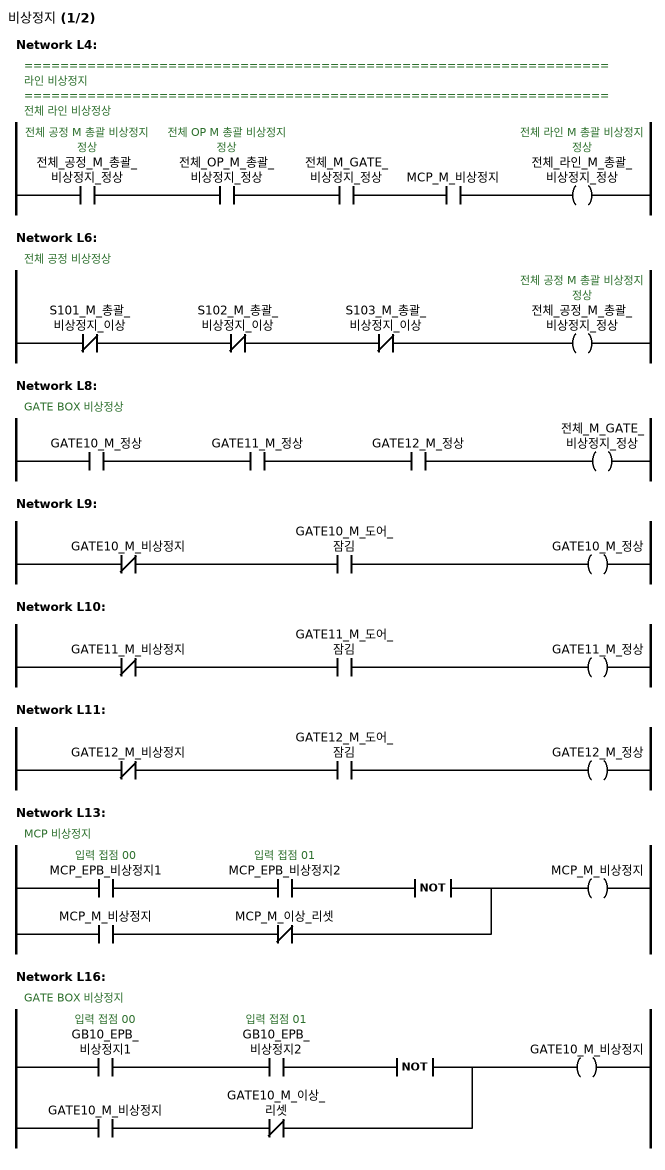
(* ================================================================= *)
(* 라인 비상정지 *)
(* ================================================================= *)
(* 전체 라인 비상정상 *)
(* Rung L4 *)
전체_라인_M_총괄_비상정지_정상 := 전체_공정_M_총괄_비상정지_정상 AND 전체_OP_M_총괄_비상정지_정상 AND 전체_M_GATE_비상정지_정상 AND MCP_M_비상정지;
(* 전체 공정 비상정상 *)
(* Rung L6 *)
전체_공정_M_총괄_비상정지_정상 := NOT S101_M_총괄_비상정지_이상 AND NOT S102_M_총괄_비상정지_이상 AND NOT S103_M_총괄_비상정지_이상;
(* GATE BOX 비상정상 *)
(* Rung L8 *)
전체_M_GATE_비상정지_정상 := GATE10_M_정상 AND GATE11_M_정상 AND GATE12_M_정상;
(* Rung L9 *)
GATE10_M_정상 := NOT GATE10_M_비상정지 AND GATE10_M_도어_잠김;
(* Rung L10 *)
GATE11_M_정상 := NOT GATE11_M_비상정지 AND GATE11_M_도어_잠김;
(* Rung L11 *)
GATE12_M_정상 := NOT GATE12_M_비상정지 AND GATE12_M_도어_잠김;
(* MCP 비상정지 *)
(* Rung L13 *)
MCP_M_비상정지 := NOT (MCP_EPB_비상정지1 AND MCP_EPB_비상정지2) OR (MCP_M_비상정지 AND NOT MCP_M_이상_리셋);
(* GATE BOX 비상정지 *)
(* Rung L16 *)
GATE10_M_비상정지 := NOT (GB10_EPB_비상정지1 AND GB10_EPB_비상정지2) OR (GATE10_M_비상정지 AND NOT GATE10_M_이상_리셋);

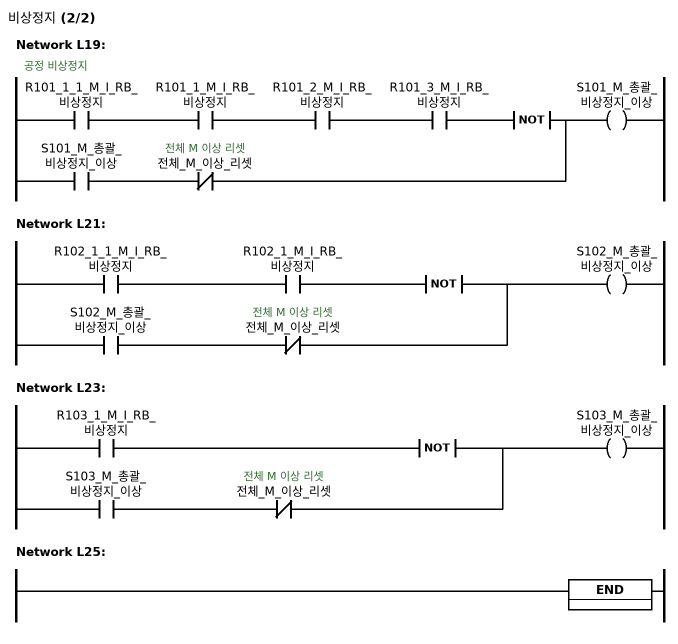
(* 공정 비상정지 *)
(* Rung L19 *)
S101_M_총괄_비상정지_이상 := NOT (R101_1_1_M_I_RB_비상정지 AND R101_1_M_I_RB_비상정지 AND R101_2_M_I_RB_비상정지 AND R101_3_M_I_RB_비상정지) OR (S101_M_총괄_비상정지_이상 AND NOT 전체_M_이상_리셋);
(* Rung L21 *)
S102_M_총괄_비상정지_이상 := NOT (R102_1_1_M_I_RB_비상정지 AND R102_1_M_I_RB_비상정지) OR (S102_M_총괄_비상정지_이상 AND NOT 전체_M_이상_리셋);
(* Rung L23 *)
S103_M_총괄_비상정지_이상 := NOT R103_1_M_I_RB_비상정지 OR (S103_M_총괄_비상정지_이상 AND NOT 전체_M_이상_리셋);
(* Rung L25 *)
END();
END_PROGRAM

PROGRAM S101_유틸리티 (* task: 스캔 프로그램 *)
VAR_EXTERNAL
    AWAYS_ON : BOOL; (* AT %MW3.1 *)
    EGIS_EJS : BOOL;
    MCP_PBL_101_자동_운전 : BOOL; (* AT %MW87630.4 *) (* 입력 접점 04 *)
    MCP_PBL_운전준비_ON : BOOL; (* AT %MW87630.0 *) (* 입력 접점 00 *)
    MCP_SSP_101_수동_선택 : BOOL; (* AT %MW87630.2 *) (* 입력 접점 02 *)
    MCP_SSP_101_자동_선택 : BOOL; (* AT %MW87630.3 *) (* 입력 접점 03 *)
    R101_1_1_M_I_RB_2차_작업완료 : BOOL; (* AT %MW20041.3 *)
    R101_1_1_M_I_RB_간섭무_1 : BOOL; (* AT %MW20042.0 *)
    R101_1_1_M_I_RB_간섭무_2 : BOOL; (* AT %MW20042.1 *)
    R101_1_1_M_I_RB_원위치 : BOOL; (* AT %MW20040.3 *)
    R101_1_1_M_SEQ : WORD; (* AT %MW10000 *) (* R101_1_1_M_SEQ *)
    R101_1_1_M_STN_차종_NONE : BOOL; (* AT %MW1002.3 *)
    R101_1_1_M_STN_차종_ON : BOOL; (* AT %MW1002.2 *)
    R101_1_1_M_차종1_AX : BOOL; (* AT %MW10001.0 *) (* R101_1_1_M_차종1_AX *)
    R101_1_1_M_차종1_B : BOOL; (* AT %MW10001.1 *) (* R101_1_1_M_차종1_B *)
    R101_1_1_M_차종1_C : BOOL; (* AT %MW10001.2 *) (* R101_1_1_M_차종1_C *)
    R101_1_1_M_차종1_D : BOOL; (* AT %MW10001.3 *) (* R101_1_1_M_차종1_D *)
    R101_1_1_M_차종1_E : BOOL; (* AT %MW10001.4 *) (* R101_1_1_M_차종1_E *)
    R101_1_1_M_차종1_F : BOOL; (* AT %MW10001.5 *) (* R101_1_1_M_차종1_F *)
    R101_1_1_M_차종1_G : BOOL; (* AT %MW10001.6 *) (* R101_1_1_M_차종1_G *)
    R101_1_1_M_차종1_H : BOOL; (* AT %MW10001.7 *) (* R101_1_1_M_차종1_H *)
    R101_1_1_M_차종2_3DR : BOOL; (* AT %MW10001.8 *) (* R101_1_1_M_차종2_3DR *)
    R101_1_1_M_차종2_4DR : BOOL; (* AT %MW10001.9 *) (* R101_1_1_M_차종2_4DR *)
    R101_1_1_M_차종2_5DR : BOOL; (* AT %MW10001.10 *) (* R101_1_1_M_차종2_5DR *)
    R101_1_1_M_차종2_SP1 : BOOL; (* AT %MW10001.12 *) (* R101_1_1_M_차종2_SP1 *)
    R101_1_1_M_차종2_SP2 : BOOL; (* AT %MW10001.13 *) (* R101_1_1_M_차종2_SP2 *)
    R101_1_1_M_차종2_WGN : BOOL; (* AT %MW10001.11 *) (* R101_1_1_M_차종2_WGN *)
    R101_1_1_M_차종3_LHD : BOOL; (* AT %MW10001.14 *) (* R101_1_1_M_차종3_LHD *)
    R101_1_1_M_차종3_RHD : BOOL; (* AT %MW10001.15 *) (* R101_1_1_M_차종3_RHD *)
    R101_1_1_M_차종4_EEC : BOOL; (* AT %MW10002.3 *) (* R101_1_1_M_차종4_EEC *)
    R101_1_1_M_차종4_SP1 : BOOL; (* AT %MW10002.8 *) (* R101_1_1_M_차종4_SP1 *)
    R101_1_1_M_차종4_SP2 : BOOL; (* AT %MW10002.9 *) (* R101_1_1_M_차종4_SP2 *)
    R101_1_1_M_차종4_SP3 : BOOL; (* AT %MW10002.11 *) (* R101_1_1_M_차종4_SP3 *)
    R101_1_1_M_차종4_SP4 : BOOL; (* AT %MW10002.12 *) (* R101_1_1_M_차종4_SP4 *)
    R101_1_1_M_차종4_SP5 : BOOL; (* AT %MW10002.13 *) (* R101_1_1_M_차종4_SP5 *)
    R101_1_1_M_차종4_SP6 : BOOL; (* AT %MW10002.14 *) (* R101_1_1_M_차종4_SP6 *)
    R101_1_1_M_차종4_SP7 : BOOL; (* AT %MW10002.15 *) (* R101_1_1_M_차종4_SP7 *)
    R101_1_1_M_차종4_내수 : BOOL; (* AT %MW10002.0 *) (* R101_1_1_M_차종4_내수 *)
    R101_1_1_M_차종4_러시아 : BOOL; (* AT %MW10002.10 *) (* R101_1_1_M_차종4_러시아 *)
    R101_1_1_M_차종4_북미 : BOOL; (* AT %MW10002.2 *) (* R101_1_1_M_차종4_북미 *)
    R101_1_1_M_차종4_브라질 : BOOL; (* AT %MW10002.7 *) (* R101_1_1_M_차종4_브라질 *)
    R101_1_1_M_차종4_수출 : BOOL; (* AT %MW10002.1 *) (* R101_1_1_M_차종4_수출 *)
    R101_1_1_M_차종4_중국 : BOOL; (* AT %MW10002.6 *) (* R101_1_1_M_차종4_중국 *)
    R101_1_1_M_차종4_중동 : BOOL; (* AT %MW10002.5 *) (* R101_1_1_M_차종4_중동 *)
    R101_1_1_M_차종4_호주 : BOOL; (* AT %MW10002.4 *) (* R101_1_1_M_차종4_호주 *)
    R101_1_1_M_차종5_AT : BOOL; (* AT %MW10003.1 *) (* R101_1_1_M_차종5_AT *)
    R101_1_1_M_차종5_MT : BOOL; (* AT %MW10003.0 *) (* R101_1_1_M_차종5_MT *)
    R101_1_1_M_차종5_SP1 : BOOL; (* AT %MW10003.2 *) (* R101_1_1_M_차종5_SP1 *)
    R101_1_1_M_차종6_DSROOF : BOOL; (* AT %MW10003.6 *) (* R101_1_1_M_차종6_DSROOF *)
    R101_1_1_M_차종6_SP1 : BOOL; (* AT %MW10003.7 *) (* R101_1_1_M_차종6_SP1 *)
    R101_1_1_M_차종6_썬루프 : BOOL; (* AT %MW10003.4 *) (* R101_1_1_M_차종6_썬루프 *)
    R101_1_1_M_차종6_일반루프 : BOOL; (* AT %MW10003.3 *) (* R101_1_1_M_차종6_일반루프 *)
    R101_1_1_M_차종6_파노라마루프 : BOOL; (* AT %MW10003.5 *) (* R101_1_1_M_차종6_파노라마루프 *)
    R101_1_1_M_차종7_DSL : BOOL; (* AT %MW10003.9 *) (* R101_1_1_M_차종7_DSL *)
    R101_1_1_M_차종7_GSL : BOOL; (* AT %MW10003.8 *) (* R101_1_1_M_차종7_GSL *)
    R101_1_1_M_차종7_SP1 : BOOL; (* AT %MW10003.10 *) (* R101_1_1_M_차종7_SP1 *)
    R101_1_1_M_차종7_SP2 : BOOL; (* AT %MW10003.11 *) (* R101_1_1_M_차종7_SP2 *)
    R101_1_1_M_차종7_SP3 : BOOL; (* AT %MW10003.12 *) (* R101_1_1_M_차종7_SP3 *)
    R101_1_1_M_차종7_SP4 : BOOL; (* AT %MW10003.13 *) (* R101_1_1_M_차종7_SP4 *)
    R101_1_1_M_차종7_SP5 : BOOL; (* AT %MW10003.14 *) (* R101_1_1_M_차종7_SP5 *)
    R101_1_1_M_차종7_SP6 : BOOL; (* AT %MW10003.15 *) (* R101_1_1_M_차종7_SP6 *)
    R101_1_1_M_차종8_2WD : BOOL; (* AT %MW10004.0 *) (* R101_1_1_M_차종8_2WD *)
    R101_1_1_M_차종8_4WD : BOOL; (* AT %MW10004.1 *) (* R101_1_1_M_차종8_4WD *)
    R101_1_1_M_차종8_SP1 : BOOL; (* AT %MW10004.2 *) (* R101_1_1_M_차종8_SP1 *)
    R101_1_1_M_차종9_MPI : BOOL; (* AT %MW10004.3 *) (* R101_1_1_M_차종9_MPI *)
    R101_1_1_M_차종9_SP1 : BOOL; (* AT %MW10004.5 *) (* R101_1_1_M_차종9_SP1 *)
    R101_1_1_M_차종9_SP10 : BOOL; (* AT %MW10004.14 *) (* R101_1_1_M_차종9_SP10 *)
    R101_1_1_M_차종9_SP11 : BOOL; (* AT %MW10004.15 *) (* R101_1_1_M_차종9_SP11 *)
    R101_1_1_M_차종9_SP2 : BOOL; (* AT %MW10004.6 *) (* R101_1_1_M_차종9_SP2 *)
    R101_1_1_M_차종9_SP3 : BOOL; (* AT %MW10004.7 *) (* R101_1_1_M_차종9_SP3 *)
    R101_1_1_M_차종9_SP4 : BOOL; (* AT %MW10004.8 *) (* R101_1_1_M_차종9_SP4 *)
    R101_1_1_M_차종9_SP5 : BOOL; (* AT %MW10004.9 *) (* R101_1_1_M_차종9_SP5 *)
    R101_1_1_M_차종9_SP6 : BOOL; (* AT %MW10004.10 *) (* R101_1_1_M_차종9_SP6 *)
    R101_1_1_M_차종9_SP7 : BOOL; (* AT %MW10004.11 *) (* R101_1_1_M_차종9_SP7 *)
    R101_1_1_M_차종9_SP8 : BOOL; (* AT %MW10004.12 *) (* R101_1_1_M_차종9_SP8 *)
    R101_1_1_M_차종9_SP9 : BOOL; (* AT %MW10004.13 *) (* R101_1_1_M_차종9_SP9 *)
    R101_1_1_M_차종9_T_GDI : BOOL; (* AT %MW10004.4 *) (* R101_1_1_M_차종9_T_GDI *)
    R101_1_1_M_차종_OPT1_R_RACK_무 : BOOL; (* AT %MW10005.3 *) (* R101_1_1_M_차종_OPT1_R_RACK_무 *)
    R101_1_1_M_차종_OPT1_R_RACK_유 : BOOL; (* AT %MW10005.2 *) (* R101_1_1_M_차종_OPT1_R_RACK_유 *)
    R101_1_1_M_차종_OPT1_SP1 : BOOL; (* AT %MW10005.10 *) (* R101_1_1_M_차종_OPT1_SP1 *)
    R101_1_1_M_차종_OPT1_SP2 : BOOL; (* AT %MW10005.11 *) (* R101_1_1_M_차종_OPT1_SP2 *)
    R101_1_1_M_차종_OPT1_SP3 : BOOL; (* AT %MW10005.12 *) (* R101_1_1_M_차종_OPT1_SP3 *)
    R101_1_1_M_차종_OPT1_SP4 : BOOL; (* AT %MW10005.13 *) (* R101_1_1_M_차종_OPT1_SP4 *)
    R101_1_1_M_차종_OPT1_SP5 : BOOL; (* AT %MW10005.14 *) (* R101_1_1_M_차종_OPT1_SP5 *)
    R101_1_1_M_차종_OPT1_SP6 : BOOL; (* AT %MW10005.15 *) (* R101_1_1_M_차종_OPT1_SP6 *)
    R101_1_1_M_차종_OPT1_S_REP_EATER_무 : BOOL; (* AT %MW10005.7 *) (* R101_1_1_M_차종_OPT1_S_REP_EATER_무 *)
    R101_1_1_M_차종_OPT1_S_REP_EATER_유 : BOOL; (* AT %MW10005.6 *) (* R101_1_1_M_차종_OPT1_S_REP_EATER_유 *)
    R101_1_1_M_차종_OPT1_VAN_무 : BOOL; (* AT %MW10005.9 *) (* R101_1_1_M_차종_OPT1_VAN_무 *)
    R101_1_1_M_차종_OPT1_VAN_유 : BOOL; (* AT %MW10005.8 *) (* R101_1_1_M_차종_OPT1_VAN_유 *)
    R101_1_1_M_차종_OPT1_슬라이딩_무 : BOOL; (* AT %MW10005.1 *) (* R101_1_1_M_차종_OPT1_슬라이딩_무 *)
    R101_1_1_M_차종_OPT1_슬라이딩_유 : BOOL; (* AT %MW10005.0 *) (* R101_1_1_M_차종_OPT1_슬라이딩_유 *)
    R101_1_1_M_차종_OPT1_폴딩_무 : BOOL; (* AT %MW10005.5 *) (* R101_1_1_M_차종_OPT1_폴딩_무 *)
    R101_1_1_M_차종_OPT1_폴딩_유 : BOOL; (* AT %MW10005.4 *) (* R101_1_1_M_차종_OPT1_폴딩_유 *)
    R101_1_M_I_RB_간섭무_2 : BOOL; (* AT %MW20072.1 *)
    R101_1_M_I_RB_원위치 : BOOL; (* AT %MW20070.3 *)
    R101_1_M_I_RB_최종작업완료 : BOOL; (* AT %MW20071.0 *)
    R101_1_M_RB_PROG_NO : WORD; (* AT %MW20074 *)
    R101_2_M_I_RB_간섭무_2 : BOOL; (* AT %MW20062.1 *)
    R101_2_M_I_RB_원위치 : BOOL; (* AT %MW20060.3 *)
    R101_2_M_I_RB_최종작업완료 : BOOL; (* AT %MW20061.0 *)
    R101_3_M_I_RB_간섭무_2 : BOOL; (* AT %MW20052.1 *)
    R101_3_M_I_RB_원위치 : BOOL; (* AT %MW20050.3 *)
    R102_1_M_I_RB_2차_작업완료 : BOOL; (* AT %MW20081.3 *)
    R102_1_M_I_RB_3차_작업완료 : BOOL; (* AT %MW20081.4 *)
    R102_1_M_I_RB_4차_작업완료 : BOOL; (* AT %MW20081.5 *)
    R102_1_M_I_RB_간섭무_1 : BOOL; (* AT %MW20082.0 *)
    R102_1_M_I_RB_간섭무_2 : BOOL; (* AT %MW20082.1 *)
    R102_1_M_I_RB_간섭무_3 : BOOL; (* AT %MW20082.2 *)
    R102_1_M_I_RB_원위치 : BOOL; (* AT %MW20080.3 *)
    R103_1_M_I_RB_최종작업완료 : BOOL; (* AT %MW20101.0 *)
    S101_3축_1_운전준비1 : BOOL; (* AT %MW50000.0 *)
    S101_3축_1_운전준비2 : BOOL; (* AT %MW50000.1 *)
    S101_3축_1_이상_리셋 : BOOL; (* AT %MW51000.7 *)
    S101_3축_2_운전준비1 : BOOL; (* AT %MW50100.0 *)
    S101_3축_2_운전준비2 : BOOL; (* AT %MW50100.1 *)
    S101_3축_2_이상_리셋 : BOOL; (* AT %MW51100.7 *)
    S101_3축_3_FAULT : BOOL; (* AT %MW50200.3 *)
    S101_3축_3_운전준비1 : BOOL; (* AT %MW50200.0 *)
    S101_3축_3_운전준비2 : BOOL; (* AT %MW50200.1 *)
    S101_3축_3_이상_리셋 : BOOL; (* AT %MW51200.7 *)
    S101_MCR_비상정지1 : BOOL; (* AT %MW95207.0 *) (* 출력 접점 00 *)
    S101_MCR_비상정지2 : BOOL; (* AT %MW95207.1 *) (* 출력 접점 01 *)
    S101_MCR_비상정지3 : BOOL; (* AT %MW95207.2 *) (* 출력 접점 02 *)
    S101_M_3_축1_전진단 : BOOL; (* AT %MW1102.3 *)
    S101_M_3_축1_후진단 : BOOL; (* AT %MW1102.4 *)
    S101_M_3_축2_전진단 : BOOL; (* AT %MW1103.3 *)
    S101_M_3_축2_후진단 : BOOL; (* AT %MW1103.4 *)
    S101_M_3_축3_전진단 : BOOL; (* AT %MW1104.3 *)
    S101_M_3_축3_후진단 : BOOL; (* AT %MW1104.4 *)
    S101_M_APRON_LH_안착OK_POS : BOOL; (* AT %MW1004.8 *)
    S101_M_APRON_RH_안착OK_POS : BOOL; (* AT %MW1004.9 *)
    S101_M_AX_래치_전진단 : BOOL; (* AT %MW1100.3 *)
    S101_M_AX_래치_후진단 : BOOL; (* AT %MW1100.4 *)
    S101_M_DASH_안착OK_POS : BOOL; (* AT %MW1004.10 *)
    S101_M_DASH_클램프_전진단 : BOOL; (* AT %MW1105.3 *)
    S101_M_DASH_클램프_후진단 : BOOL; (* AT %MW1105.4 *)
    S101_M_FRT_취출OK_POS : BOOL; (* AT %MW1004.11 *)
    S101_M_SEQ : WORD; (* AT %MW10020 *) (* S101_M_SEQ *)
    S101_M_SHIFT_전진단 : BOOL; (* AT %MW1101.3 *)
    S101_M_SHIFT_후진단 : BOOL; (* AT %MW1101.4 *)
    S101_M_STN_DASH_로딩완료 : BOOL; (* AT %MW1001.12 *)
    S101_M_STN_FRT_FLR_취출완료 : BOOL; (* AT %MW1001.13 *)
    S101_M_STN_LH_로딩완료 : BOOL; (* AT %MW1001.10 *)
    S101_M_STN_RH_로딩완료 : BOOL; (* AT %MW1001.11 *)
    S101_M_STN_차종_NONE : BOOL; (* AT %MW1002.1 *)
    S101_M_STN_차종_ON : BOOL; (* AT %MW1002.0 *)
    S101_M_공정_APRON_제품감지_OFF : BOOL; (* AT %MW1001.4 *)
    S101_M_공정_APRON_제품감지_ON : BOOL; (* AT %MW1001.3 *)
    S101_M_공정_DASH_제품감지_OFF : BOOL; (* AT %MW1001.6 *)
    S101_M_공정_DASH_제품감지_ON : BOOL; (* AT %MW1001.5 *)
    S101_M_공정_HOME_POSI : BOOL; (* AT %MW1004.0 *)
    S101_M_공정_간섭무 : BOOL; (* AT %MW1004.1 *)
    S101_M_공정_사양감지_OK : BOOL; (* AT %MW1001.7 *)
    S101_M_사양이상 : BOOL; (* AT %MW1019.0 *)
    S101_M_수동_모드 : BOOL; (* AT %MW1000.3 *)
    S101_M_운전준비_ON : BOOL; (* AT %MW1000.0 *)
    S101_M_자동_START : BOOL; (* AT %MW1000.5 *)
    S101_M_자동_모드 : BOOL; (* AT %MW1000.1 *)
    S101_M_자동_운전중 : BOOL; (* AT %MW1000.4 *)
    S101_M_작업_완료 : BOOL; (* AT %MW1001.0 *)
    S101_M_작업_완료_보조 : BOOL; (* AT %MW1000.9 *)
    S101_M_전체_클램프_잠김단 : BOOL; (* AT %MW1004.12 *)
    S101_M_차종1_AX : BOOL; (* AT %MW10021.0 *) (* S101_M_차종1_AX *)
    S101_M_차종1_B : BOOL; (* AT %MW10021.1 *) (* S101_M_차종1_B *)
    S101_M_차종1_C : BOOL; (* AT %MW10021.2 *) (* S101_M_차종1_C *)
    S101_M_차종1_D : BOOL; (* AT %MW10021.3 *) (* S101_M_차종1_D *)
    S101_M_차종1_E : BOOL; (* AT %MW10021.4 *) (* S101_M_차종1_E *)
    S101_M_차종1_F : BOOL; (* AT %MW10021.5 *) (* S101_M_차종1_F *)
    S101_M_차종1_G : BOOL; (* AT %MW10021.6 *) (* S101_M_차종1_G *)
    S101_M_차종1_H : BOOL; (* AT %MW10021.7 *) (* S101_M_차종1_H *)
    S101_M_차종2_3DR : BOOL; (* AT %MW10021.8 *) (* S101_M_차종2_3DR *)
    S101_M_차종2_4DR : BOOL; (* AT %MW10021.9 *) (* S101_M_차종2_4DR *)
    S101_M_차종2_5DR : BOOL; (* AT %MW10021.10 *) (* S101_M_차종2_5DR *)
    S101_M_차종2_SP1 : BOOL; (* AT %MW10021.12 *) (* S101_M_차종2_SP1 *)
    S101_M_차종2_SP2 : BOOL; (* AT %MW10021.13 *) (* S101_M_차종2_SP2 *)
    S101_M_차종2_WGN : BOOL; (* AT %MW10021.11 *) (* S101_M_차종2_WGN *)
    S101_M_차종3_LHD : BOOL; (* AT %MW10021.14 *) (* S101_M_차종3_LHD *)
    S101_M_차종3_RHD : BOOL; (* AT %MW10021.15 *) (* S101_M_차종3_RHD *)
    S101_M_차종4_EEC : BOOL; (* AT %MW10022.3 *) (* S101_M_차종4_EEC *)
    S101_M_차종4_SP1 : BOOL; (* AT %MW10022.8 *) (* S101_M_차종4_SP1 *)
    S101_M_차종4_SP2 : BOOL; (* AT %MW10022.9 *) (* S101_M_차종4_SP2 *)
    S101_M_차종4_SP3 : BOOL; (* AT %MW10022.11 *) (* S101_M_차종4_SP3 *)
    S101_M_차종4_SP4 : BOOL; (* AT %MW10022.12 *) (* S101_M_차종4_SP4 *)
    S101_M_차종4_SP5 : BOOL; (* AT %MW10022.13 *) (* S101_M_차종4_SP5 *)
    S101_M_차종4_SP6 : BOOL; (* AT %MW10022.14 *) (* S101_M_차종4_SP6 *)
    S101_M_차종4_SP7 : BOOL; (* AT %MW10022.15 *) (* S101_M_차종4_SP7 *)
    S101_M_차종4_내수 : BOOL; (* AT %MW10022.0 *) (* S101_M_차종4_내수 *)
    S101_M_차종4_러시아 : BOOL; (* AT %MW10022.10 *) (* S101_M_차종4_러시아 *)
    S101_M_차종4_북미 : BOOL; (* AT %MW10022.2 *) (* S101_M_차종4_북미 *)
    S101_M_차종4_브라질 : BOOL; (* AT %MW10022.7 *) (* S101_M_차종4_브라질 *)
    S101_M_차종4_수출 : BOOL; (* AT %MW10022.1 *) (* S101_M_차종4_수출 *)
    S101_M_차종4_중국 : BOOL; (* AT %MW10022.6 *) (* S101_M_차종4_중국 *)
    S101_M_차종4_중동 : BOOL; (* AT %MW10022.5 *) (* S101_M_차종4_중동 *)
    S101_M_차종4_호주 : BOOL; (* AT %MW10022.4 *) (* S101_M_차종4_호주 *)
    S101_M_차종5_AT : BOOL; (* AT %MW10023.1 *) (* S101_M_차종5_AT *)
    S101_M_차종5_MT : BOOL; (* AT %MW10023.0 *) (* S101_M_차종5_MT *)
    S101_M_차종5_SP1 : BOOL; (* AT %MW10023.2 *) (* S101_M_차종5_SP1 *)
    S101_M_차종6_DSROOF : BOOL; (* AT %MW10023.6 *) (* S101_M_차종6_DSROOF *)
    S101_M_차종6_SP1 : BOOL; (* AT %MW10023.7 *) (* S101_M_차종6_SP1 *)
    S101_M_차종6_썬루프 : BOOL; (* AT %MW10023.4 *) (* S101_M_차종6_썬루프 *)
    S101_M_차종6_일반루프 : BOOL; (* AT %MW10023.3 *) (* S101_M_차종6_일반루프 *)
    S101_M_차종6_파노라마루프 : BOOL; (* AT %MW10023.5 *) (* S101_M_차종6_파노라마루프 *)
    S101_M_차종7_DSL : BOOL; (* AT %MW10023.9 *) (* S101_M_차종7_DSL *)
    S101_M_차종7_GSL : BOOL; (* AT %MW10023.8 *) (* S101_M_차종7_GSL *)
    S101_M_차종7_SP1 : BOOL; (* AT %MW10023.10 *) (* S101_M_차종7_SP1 *)
    S101_M_차종7_SP2 : BOOL; (* AT %MW10023.11 *) (* S101_M_차종7_SP2 *)
    S101_M_차종7_SP3 : BOOL; (* AT %MW10023.12 *) (* S101_M_차종7_SP3 *)
    S101_M_차종7_SP4 : BOOL; (* AT %MW10023.13 *) (* S101_M_차종7_SP4 *)
    S101_M_차종7_SP5 : BOOL; (* AT %MW10023.14 *) (* S101_M_차종7_SP5 *)
    S101_M_차종7_SP6 : BOOL; (* AT %MW10023.15 *) (* S101_M_차종7_SP6 *)
    S101_M_차종8_2WD : BOOL; (* AT %MW10024.0 *) (* S101_M_차종8_2WD *)
    S101_M_차종8_4WD : BOOL; (* AT %MW10024.1 *) (* S101_M_차종8_4WD *)
    S101_M_차종8_SP1 : BOOL; (* AT %MW10024.2 *) (* S101_M_차종8_SP1 *)
    S101_M_차종9_MPI : BOOL; (* AT %MW10024.3 *) (* S101_M_차종9_MPI *)
    S101_M_차종9_SP1 : BOOL; (* AT %MW10024.5 *) (* S101_M_차종9_SP1 *)
    S101_M_차종9_SP10 : BOOL; (* AT %MW10024.14 *) (* S101_M_차종9_SP10 *)
    S101_M_차종9_SP11 : BOOL; (* AT %MW10024.15 *) (* S101_M_차종9_SP11 *)
    S101_M_차종9_SP2 : BOOL; (* AT %MW10024.6 *) (* S101_M_차종9_SP2 *)
    S101_M_차종9_SP3 : BOOL; (* AT %MW10024.7 *) (* S101_M_차종9_SP3 *)
    S101_M_차종9_SP4 : BOOL; (* AT %MW10024.8 *) (* S101_M_차종9_SP4 *)
    S101_M_차종9_SP5 : BOOL; (* AT %MW10024.9 *) (* S101_M_차종9_SP5 *)
    S101_M_차종9_SP6 : BOOL; (* AT %MW10024.10 *) (* S101_M_차종9_SP6 *)
    S101_M_차종9_SP7 : BOOL; (* AT %MW10024.11 *) (* S101_M_차종9_SP7 *)
    S101_M_차종9_SP8 : BOOL; (* AT %MW10024.12 *) (* S101_M_차종9_SP8 *)
    S101_M_차종9_SP9 : BOOL; (* AT %MW10024.13 *) (* S101_M_차종9_SP9 *)
    S101_M_차종9_T_GDI : BOOL; (* AT %MW10024.4 *) (* S101_M_차종9_T_GDI *)
    S101_M_차종_OPT1_R_RACK_무 : BOOL; (* AT %MW10025.3 *) (* S101_M_차종_OPT1_R_RACK_무 *)
    S101_M_차종_OPT1_R_RACK_유 : BOOL; (* AT %MW10025.2 *) (* S101_M_차종_OPT1_R_RACK_유 *)
    S101_M_차종_OPT1_SP1 : BOOL; (* AT %MW10025.10 *) (* S101_M_차종_OPT1_SP1 *)
    S101_M_차종_OPT1_SP2 : BOOL; (* AT %MW10025.11 *) (* S101_M_차종_OPT1_SP2 *)
    S101_M_차종_OPT1_SP3 : BOOL; (* AT %MW10025.12 *) (* S101_M_차종_OPT1_SP3 *)
    S101_M_차종_OPT1_SP4 : BOOL; (* AT %MW10025.13 *) (* S101_M_차종_OPT1_SP4 *)
    S101_M_차종_OPT1_SP5 : BOOL; (* AT %MW10025.14 *) (* S101_M_차종_OPT1_SP5 *)
    S101_M_차종_OPT1_SP6 : BOOL; (* AT %MW10025.15 *) (* S101_M_차종_OPT1_SP6 *)
    S101_M_차종_OPT1_S_REP_EATER_무 : BOOL; (* AT %MW10025.7 *) (* S101_M_차종_OPT1_S_REP_EATER_무 *)
    S101_M_차종_OPT1_S_REP_EATER_유 : BOOL; (* AT %MW10025.6 *) (* S101_M_차종_OPT1_S_REP_EATER_유 *)
    S101_M_차종_OPT1_VAN_무 : BOOL; (* AT %MW10025.9 *) (* S101_M_차종_OPT1_VAN_무 *)
    S101_M_차종_OPT1_VAN_유 : BOOL; (* AT %MW10025.8 *) (* S101_M_차종_OPT1_VAN_유 *)
    S101_M_차종_OPT1_슬라이딩_무 : BOOL; (* AT %MW10025.1 *) (* S101_M_차종_OPT1_슬라이딩_무 *)
    S101_M_차종_OPT1_슬라이딩_유 : BOOL; (* AT %MW10025.0 *) (* S101_M_차종_OPT1_슬라이딩_유 *)
    S101_M_차종_OPT1_폴딩_무 : BOOL; (* AT %MW10025.5 *) (* S101_M_차종_OPT1_폴딩_무 *)
    S101_M_차종_OPT1_폴딩_유 : BOOL; (* AT %MW10025.4 *) (* S101_M_차종_OPT1_폴딩_유 *)
    S101_M_핀클램프_전진단 : BOOL; (* AT %MW1106.3 *)
    S101_M_핀클램프_후진단 : BOOL; (* AT %MW1106.4 *)
    S101_PRS_I_3축_DASH_파트1_ON : BOOL; (* AT %MW86102.6 *) (* 입력 접점 06 *)
    S101_PRS_I_3축_DASH_파트2_ON : BOOL; (* AT %MW86102.7 *) (* 입력 접점 07 *)
    S101_PRS_I_3축_LH_파트_ON : BOOL; (* AT %MW86102.4 *) (* 입력 접점 04 *)
    S101_PRS_I_3축_RH_파트_ON : BOOL; (* AT %MW86102.5 *) (* 입력 접점 05 *)
    S101_PRS_I_AX_APRON_LHD_사양감지 : BOOL; (* AT %MW86102.8 *)
    S101_PRS_I_AX_APRON_RHD_사양감지 : BOOL; (* AT %MW86102.9 *)
    S101_PRS_I_AX_DASH_파트_ON : BOOL; (* AT %MW86102.2 *)
    S101_PRS_I_AX_LH_파트_ON : BOOL; (* AT %MW86102.0 *)
    S101_PRS_I_AX_RH_파트_ON : BOOL; (* AT %MW86102.1 *)
    S101_운전준비 : TON;
    S103_M_공정_제품감지_ON : BOOL; (* AT %MW2001.3 *)
    T101_자동 : TON;
    전체_M_GATE_자동기동 : BOOL; (* AT %MW308.1 *) (* 전체 M GATE 자동기동 *)
    전체_M_이상_리셋 : BOOL; (* AT %MW308.2 *) (* 전체 M 이상 리셋 *)
    전체_라인_M_총괄_SAFETY_이상 : BOOL; (* AT %MW300.2 *)
    전체_라인_M_총괄_공기압_이상 : BOOL; (* AT %MW300.3 *)
    전체_라인_M_총괄_비상정지_이상 : BOOL; (* AT %MW300.1 *)
    전체_라인_M_총괄_이상 : BOOL; (* AT %MW300.0 *)
END_VAR
VAR
    _R101_1_RB_비교_PROG_NO : INT;
    작업_COMP : TON;
END_VAR
VAR
    _t1 : BOOL;
    _t2 : BOOL;
    _t3 : BOOL;
    _t4 : BOOL;
    _p5 : BOOL;
END_VAR

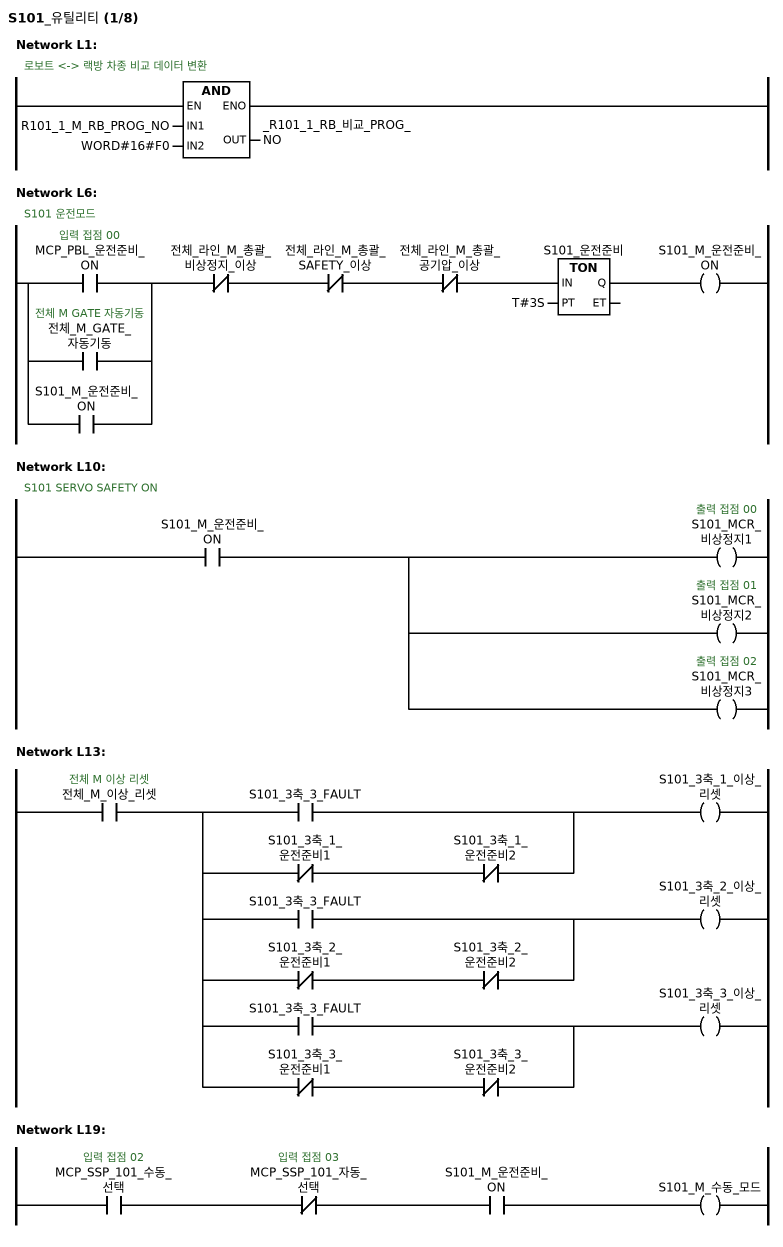
(* 로보트 <-> 랙방 차종 비교 데이터 변환 *)
(* Rung L1 *)
_R101_1_RB_비교_PROG_NO := R101_1_M_RB_PROG_NO AND WORD#16#F0;
(* S101 운전모드 *)
(* Rung L6 *)
S101_운전준비(IN := (MCP_PBL_운전준비_ON OR 전체_M_GATE_자동기동 OR S101_M_운전준비_ON) AND NOT 전체_라인_M_총괄_비상정지_이상 AND NOT 전체_라인_M_총괄_SAFETY_이상 AND NOT 전체_라인_M_총괄_공기압_이상, PT := T#3S);
S101_M_운전준비_ON := S101_운전준비.Q;
(* S101 SERVO SAFETY ON *)
(* Rung L10 *)
S101_MCR_비상정지1 := S101_M_운전준비_ON;
S101_MCR_비상정지2 := S101_M_운전준비_ON;
S101_MCR_비상정지3 := S101_M_운전준비_ON;
(* Rung L13 *)
S101_3축_1_이상_리셋 := 전체_M_이상_리셋 AND (S101_3축_3_FAULT OR (NOT S101_3축_1_운전준비1 AND NOT S101_3축_1_운전준비2));
S101_3축_2_이상_리셋 := 전체_M_이상_리셋 AND (S101_3축_3_FAULT OR (NOT S101_3축_2_운전준비1 AND NOT S101_3축_2_운전준비2));
S101_3축_3_이상_리셋 := 전체_M_이상_리셋 AND (S101_3축_3_FAULT OR (NOT S101_3축_3_운전준비1 AND NOT S101_3축_3_운전준비2));
(* Rung L19 *)
S101_M_수동_모드 := MCP_SSP_101_수동_선택 AND NOT MCP_SSP_101_자동_선택 AND S101_M_운전준비_ON;

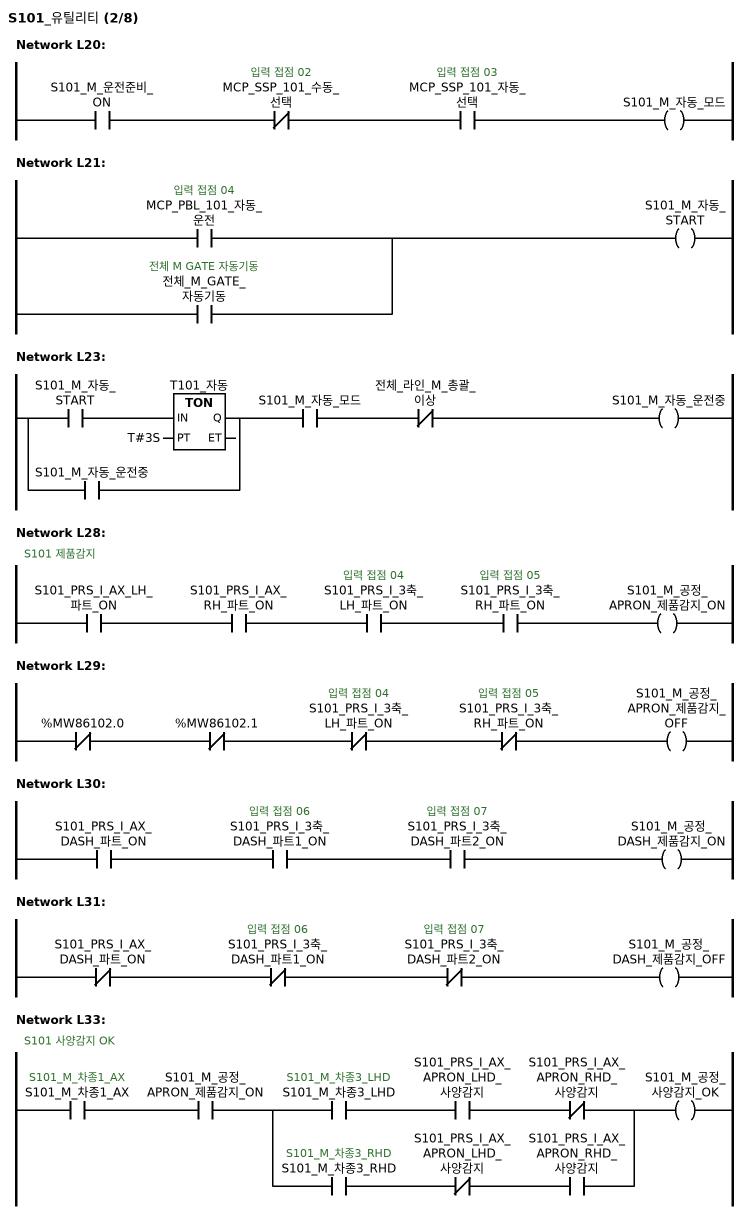
(* Rung L20 *)
S101_M_자동_모드 := S101_M_운전준비_ON AND NOT MCP_SSP_101_수동_선택 AND MCP_SSP_101_자동_선택;
(* Rung L21 *)
S101_M_자동_START := MCP_PBL_101_자동_운전 OR 전체_M_GATE_자동기동;
(* Rung L23 *)
T101_자동(IN := S101_M_자동_START, PT := T#3S);
S101_M_자동_운전중 := (T101_자동.Q OR S101_M_자동_운전중) AND S101_M_자동_모드 AND NOT 전체_라인_M_총괄_이상;
(* S101 제품감지 *)
(* Rung L28 *)
S101_M_공정_APRON_제품감지_ON := S101_PRS_I_AX_LH_파트_ON AND S101_PRS_I_AX_RH_파트_ON AND S101_PRS_I_3축_LH_파트_ON AND S101_PRS_I_3축_RH_파트_ON;
(* Rung L29 *)
S101_M_공정_APRON_제품감지_OFF := NOT %MW86102.0 AND NOT %MW86102.1 AND NOT S101_PRS_I_3축_LH_파트_ON AND NOT S101_PRS_I_3축_RH_파트_ON;
(* Rung L30 *)
S101_M_공정_DASH_제품감지_ON := S101_PRS_I_AX_DASH_파트_ON AND S101_PRS_I_3축_DASH_파트1_ON AND S101_PRS_I_3축_DASH_파트2_ON;
(* Rung L31 *)
S101_M_공정_DASH_제품감지_OFF := NOT S101_PRS_I_AX_DASH_파트_ON AND NOT S101_PRS_I_3축_DASH_파트1_ON AND NOT S101_PRS_I_3축_DASH_파트2_ON;
(* S101 사양감지 OK *)
(* Rung L33 *)
S101_M_공정_사양감지_OK := S101_M_차종1_AX AND S101_M_공정_APRON_제품감지_ON AND ((S101_M_차종3_LHD AND S101_PRS_I_AX_APRON_LHD_사양감지 AND NOT S101_PRS_I_AX_APRON_RHD_사양감지) OR (S101_M_차종3_RHD AND NOT S101_PRS_I_AX_APRON_LHD_사양감지 AND S101_PRS_I_AX_APRON_RHD_사양감지));

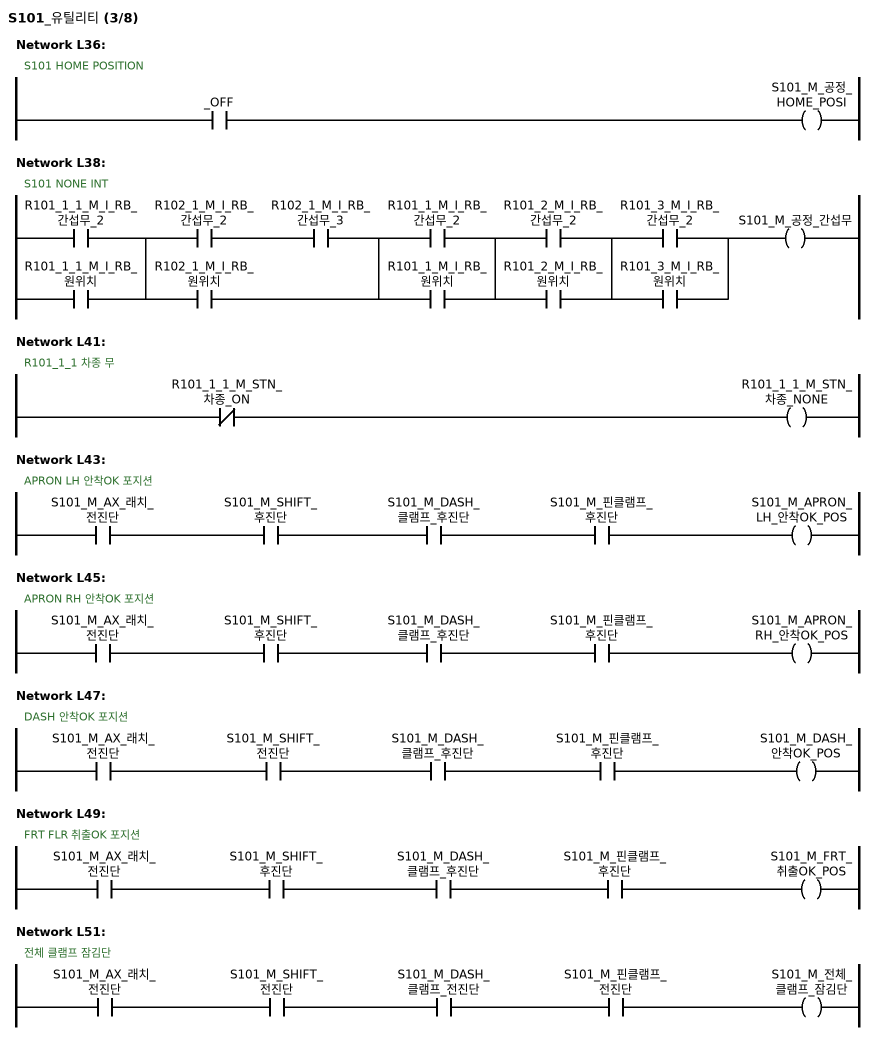
(* S101 HOME POSITION *)
(* Rung L36 *)
S101_M_공정_HOME_POSI := _OFF;
(* S101 NONE INT *)
(* Rung L38 *)
S101_M_공정_간섭무 := (R101_1_1_M_I_RB_간섭무_2 OR R101_1_1_M_I_RB_원위치) AND ((R102_1_M_I_RB_간섭무_2 AND R102_1_M_I_RB_간섭무_3) OR R102_1_M_I_RB_원위치) AND (R101_1_M_I_RB_간섭무_2 OR R101_1_M_I_RB_원위치) AND (R101_2_M_I_RB_간섭무_2 OR R101_2_M_I_RB_원위치) AND (R101_3_M_I_RB_간섭무_2 OR R101_3_M_I_RB_원위치);
(* R101_1_1 차종 무 *)
(* Rung L41 *)
R101_1_1_M_STN_차종_NONE := NOT R101_1_1_M_STN_차종_ON;
(* APRON LH 안착OK 포지션 *)
(* Rung L43 *)
S101_M_APRON_LH_안착OK_POS := S101_M_AX_래치_전진단 AND S101_M_SHIFT_후진단 AND S101_M_DASH_클램프_후진단 AND S101_M_핀클램프_후진단;
(* APRON RH 안착OK 포지션 *)
(* Rung L45 *)
S101_M_APRON_RH_안착OK_POS := S101_M_AX_래치_전진단 AND S101_M_SHIFT_후진단 AND S101_M_DASH_클램프_후진단 AND S101_M_핀클램프_후진단;
(* DASH 안착OK 포지션 *)
(* Rung L47 *)
S101_M_DASH_안착OK_POS := S101_M_AX_래치_전진단 AND S101_M_SHIFT_전진단 AND S101_M_DASH_클램프_후진단 AND S101_M_핀클램프_후진단;
(* FRT FLR 취출OK 포지션 *)
(* Rung L49 *)
S101_M_FRT_취출OK_POS := S101_M_AX_래치_전진단 AND S101_M_SHIFT_후진단 AND S101_M_DASH_클램프_후진단 AND S101_M_핀클램프_후진단;
(* 전체 클램프 잠김단 *)
(* Rung L51 *)
S101_M_전체_클램프_잠김단 := S101_M_AX_래치_전진단 AND S101_M_SHIFT_전진단 AND S101_M_DASH_클램프_전진단 AND S101_M_핀클램프_전진단;

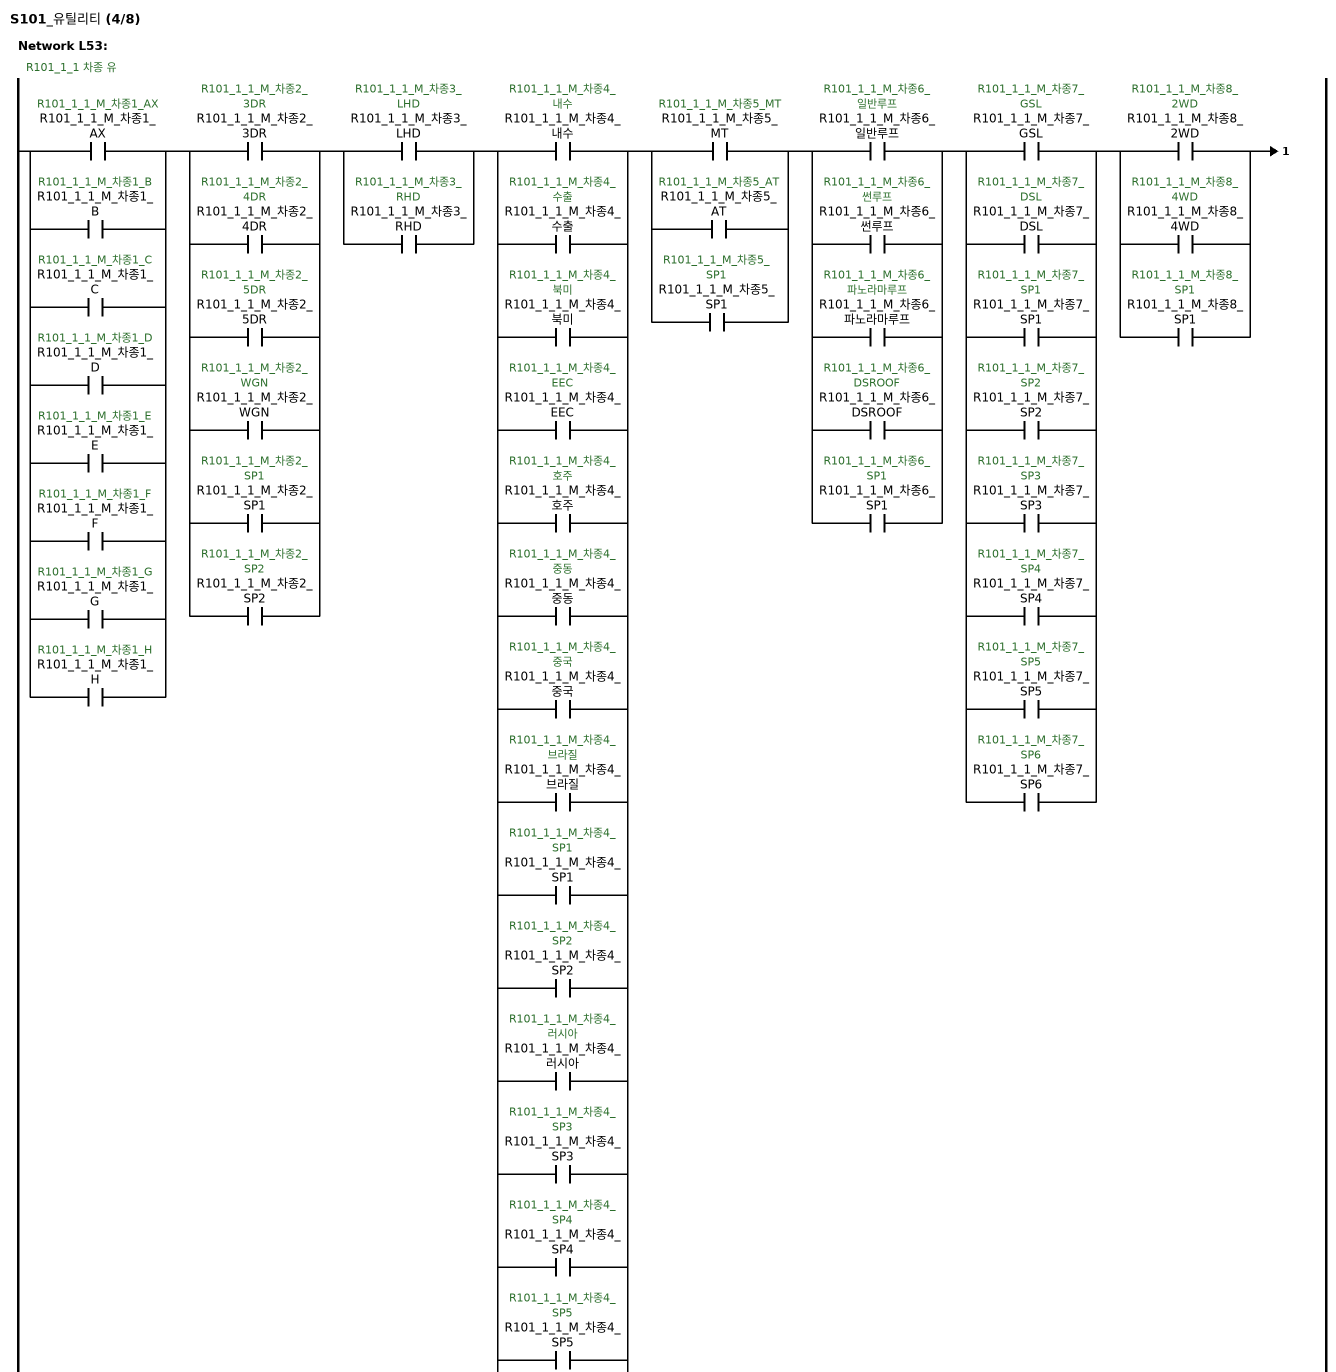

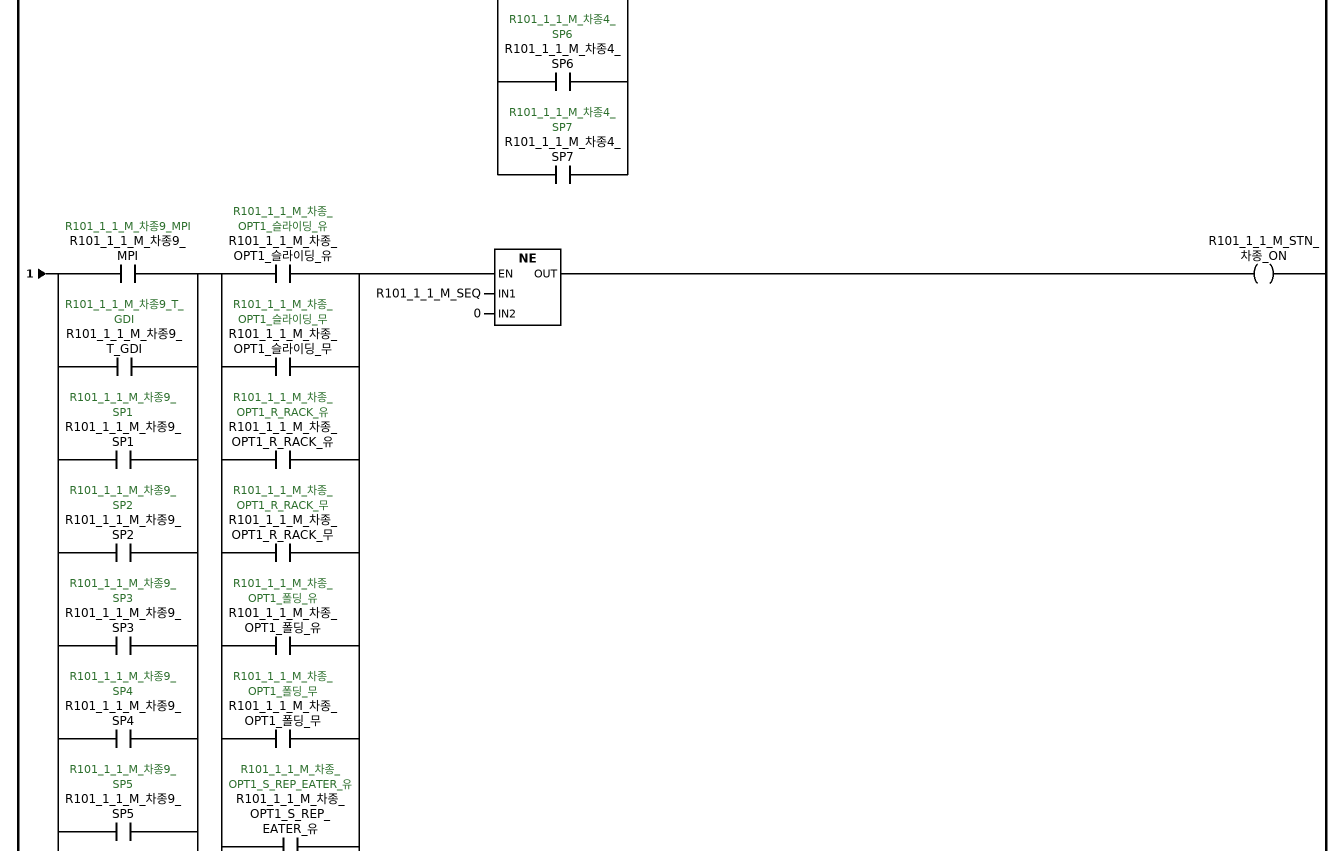

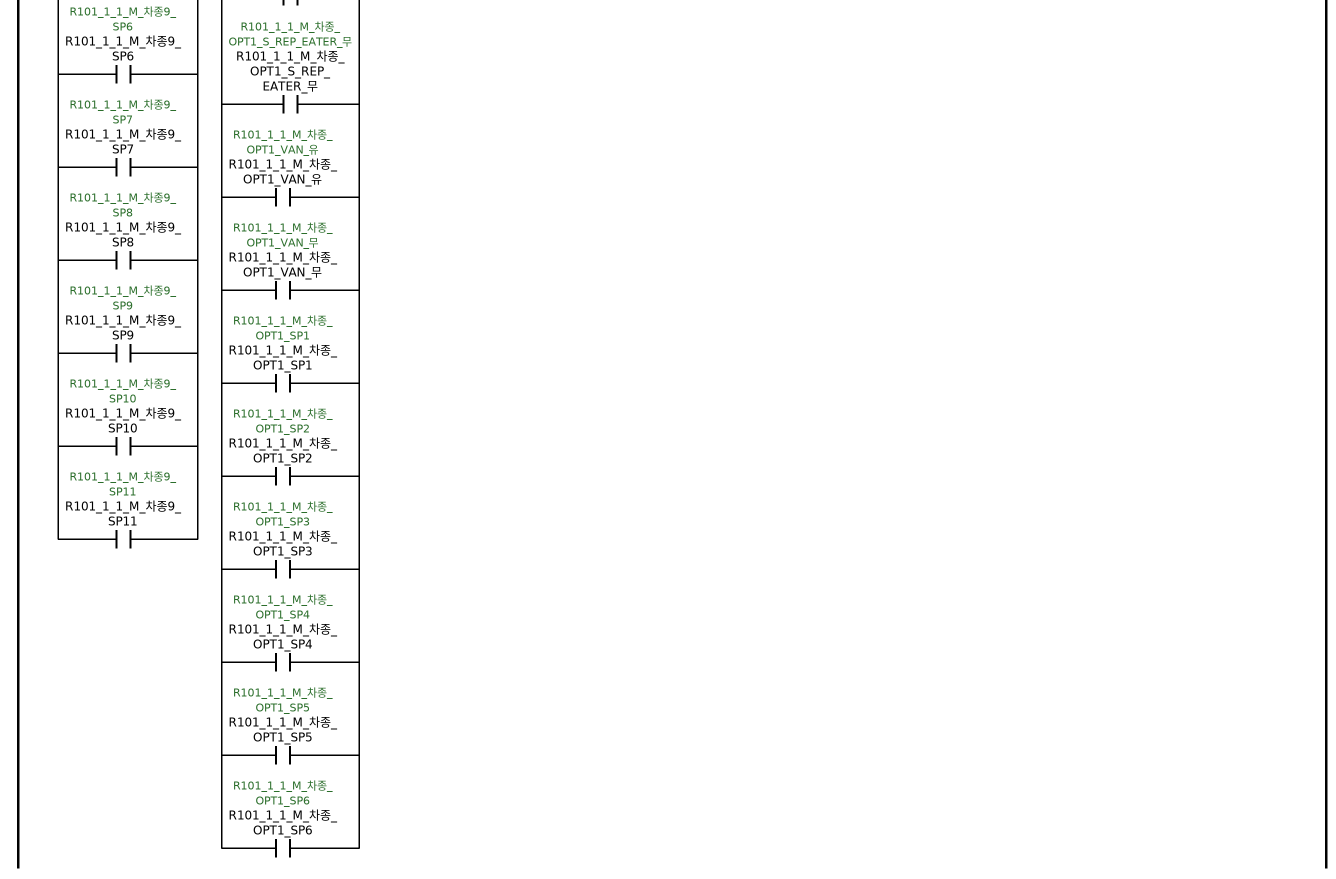
(* R101_1_1 차종 유 *)
(* Rung L53 *)
IF (R101_1_1_M_차종1_AX OR R101_1_1_M_차종1_B OR R101_1_1_M_차종1_C OR R101_1_1_M_차종1_D OR R101_1_1_M_차종1_E OR R101_1_1_M_차종1_F OR R101_1_1_M_차종1_G OR R101_1_1_M_차종1_H) AND (R101_1_1_M_차종2_3DR OR R101_1_1_M_차종2_4DR OR R101_1_1_M_차종2_5DR OR R101_1_1_M_차종2_WGN OR R101_1_1_M_차종2_SP1 OR R101_1_1_M_차종2_SP2) AND (R101_1_1_M_차종3_LHD OR R101_1_1_M_차종3_RHD) AND (R101_1_1_M_차종4_내수 OR R101_1_1_M_차종4_수출 OR R101_1_1_M_차종4_북미 OR R101_1_1_M_차종4_EEC OR R101_1_1_M_차종4_호주 OR R101_1_1_M_차종4_중동 OR R101_1_1_M_차종4_중국 OR R101_1_1_M_차종4_브라질 OR R101_1_1_M_차종4_SP1 OR R101_1_1_M_차종4_SP2 OR R101_1_1_M_차종4_러시아 OR R101_1_1_M_차종4_SP3 OR R101_1_1_M_차종4_SP4 OR R101_1_1_M_차종4_SP5 OR R101_1_1_M_차종4_SP6 OR R101_1_1_M_차종4_SP7) AND (R101_1_1_M_차종5_MT OR R101_1_1_M_차종5_AT OR R101_1_1_M_차종5_SP1) AND (R101_1_1_M_차종6_일반루프 OR R101_1_1_M_차종6_썬루프 OR R101_1_1_M_차종6_파노라마루프 OR R101_1_1_M_차종6_DSROOF OR R101_1_1_M_차종6_SP1) AND (R101_1_1_M_차종7_GSL OR R101_1_1_M_차종7_DSL OR R101_1_1_M_차종7_SP1 OR R101_1_1_M_차종7_SP2 OR R101_1_1_M_차종7_SP3 OR R101_1_1_M_차종7_SP4 OR R101_1_1_M_차종7_SP5 OR R101_1_1_M_차종7_SP6) AND (R101_1_1_M_차종8_2WD OR R101_1_1_M_차종8_4WD OR R101_1_1_M_차종8_SP1) AND (R101_1_1_M_차종9_MPI OR R101_1_1_M_차종9_T_GDI OR R101_1_1_M_차종9_SP1 OR R101_1_1_M_차종9_SP2 OR R101_1_1_M_차종9_SP3 OR R101_1_1_M_차종9_SP4 OR R101_1_1_M_차종9_SP5 OR R101_1_1_M_차종9_SP6 OR R101_1_1_M_차종9_SP7 OR R101_1_1_M_차종9_SP8 OR R101_1_1_M_차종9_SP9 OR R101_1_1_M_차종9_SP10 OR R101_1_1_M_차종9_SP11) AND (R101_1_1_M_차종_OPT1_슬라이딩_유 OR R101_1_1_M_차종_OPT1_슬라이딩_무 OR R101_1_1_M_차종_OPT1_R_RACK_유 OR R101_1_1_M_차종_OPT1_R_RACK_무 OR R101_1_1_M_차종_OPT1_폴딩_유 OR R101_1_1_M_차종_OPT1_폴딩_무 OR R101_1_1_M_차종_OPT1_S_REP_EATER_유 OR R101_1_1_M_차종_OPT1_S_REP_EATER_무 OR R101_1_1_M_차종_OPT1_VAN_유 OR R101_1_1_M_차종_OPT1_VAN_무 OR R101_1_1_M_차종_OPT1_SP1 OR R101_1_1_M_차종_OPT1_SP2 OR R101_1_1_M_차종_OPT1_SP3 OR R101_1_1_M_차종_OPT1_SP4 OR R101_1_1_M_차종_OPT1_SP5 OR R101_1_1_M_차종_OPT1_SP6) THEN
    _t1 := R101_1_1_M_SEQ <> 0;
END_IF;
R101_1_1_M_STN_차종_ON := _t1;

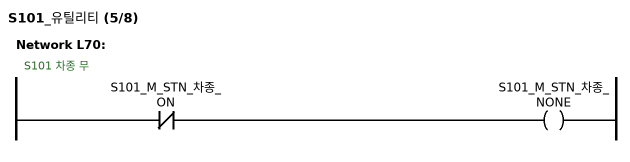
(* S101 차종 무 *)
(* Rung L70 *)
S101_M_STN_차종_NONE := NOT S101_M_STN_차종_ON;

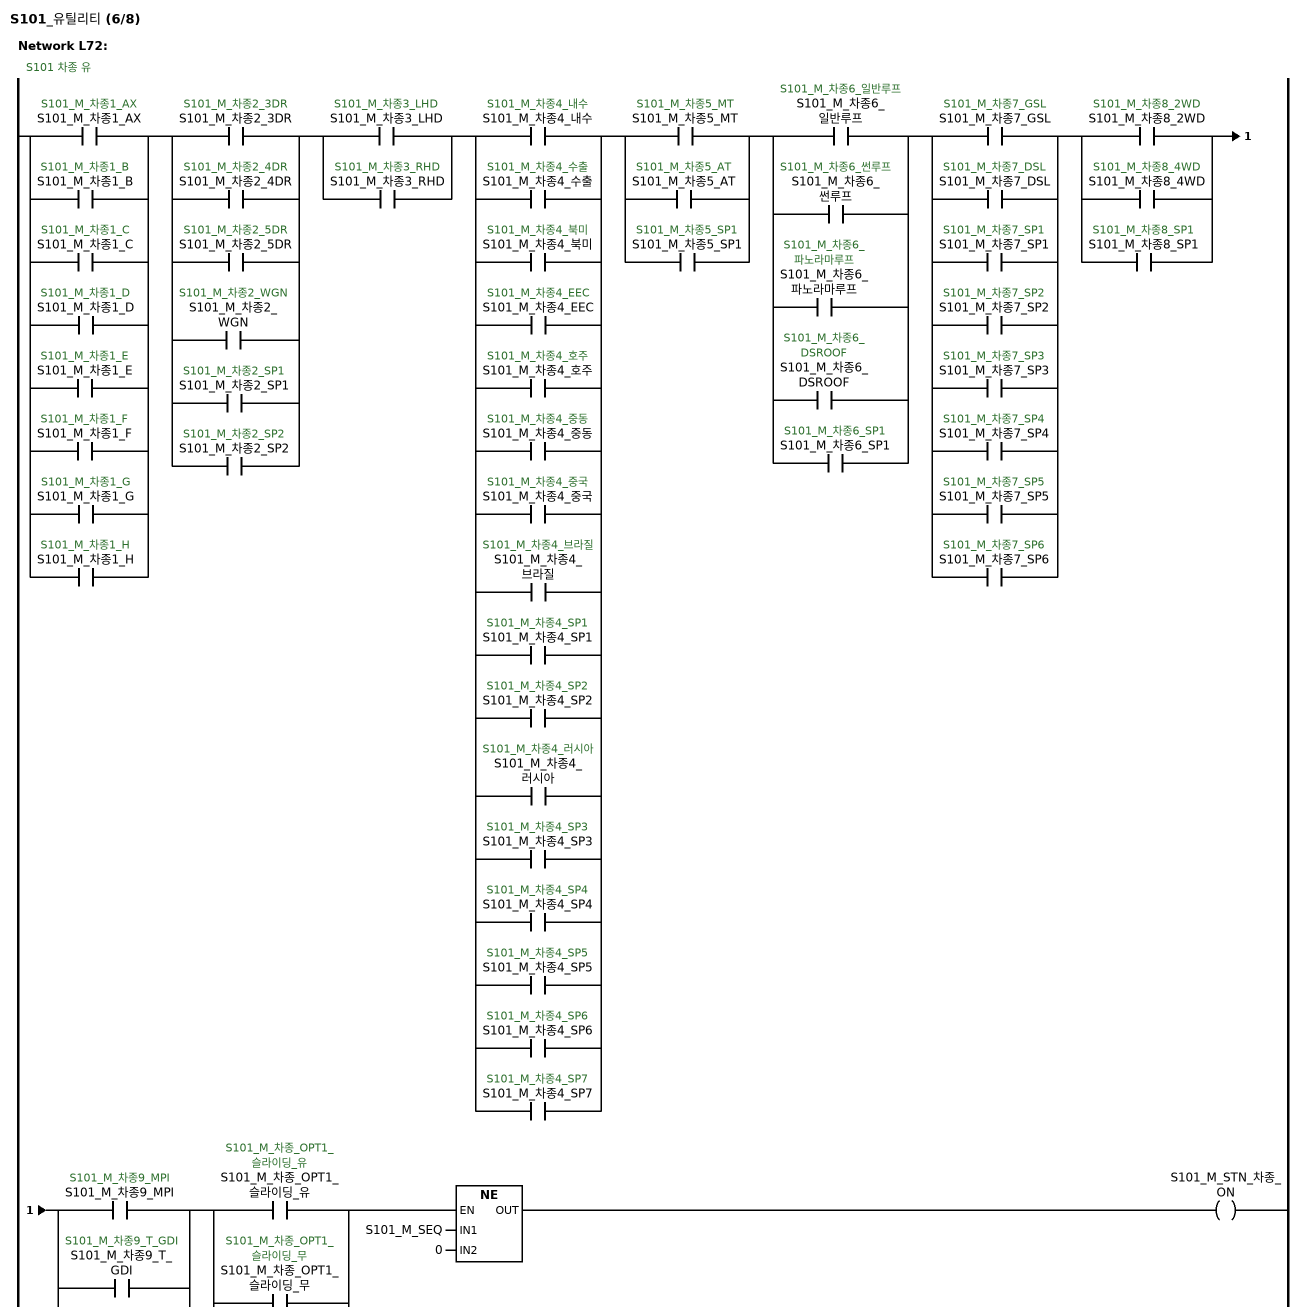

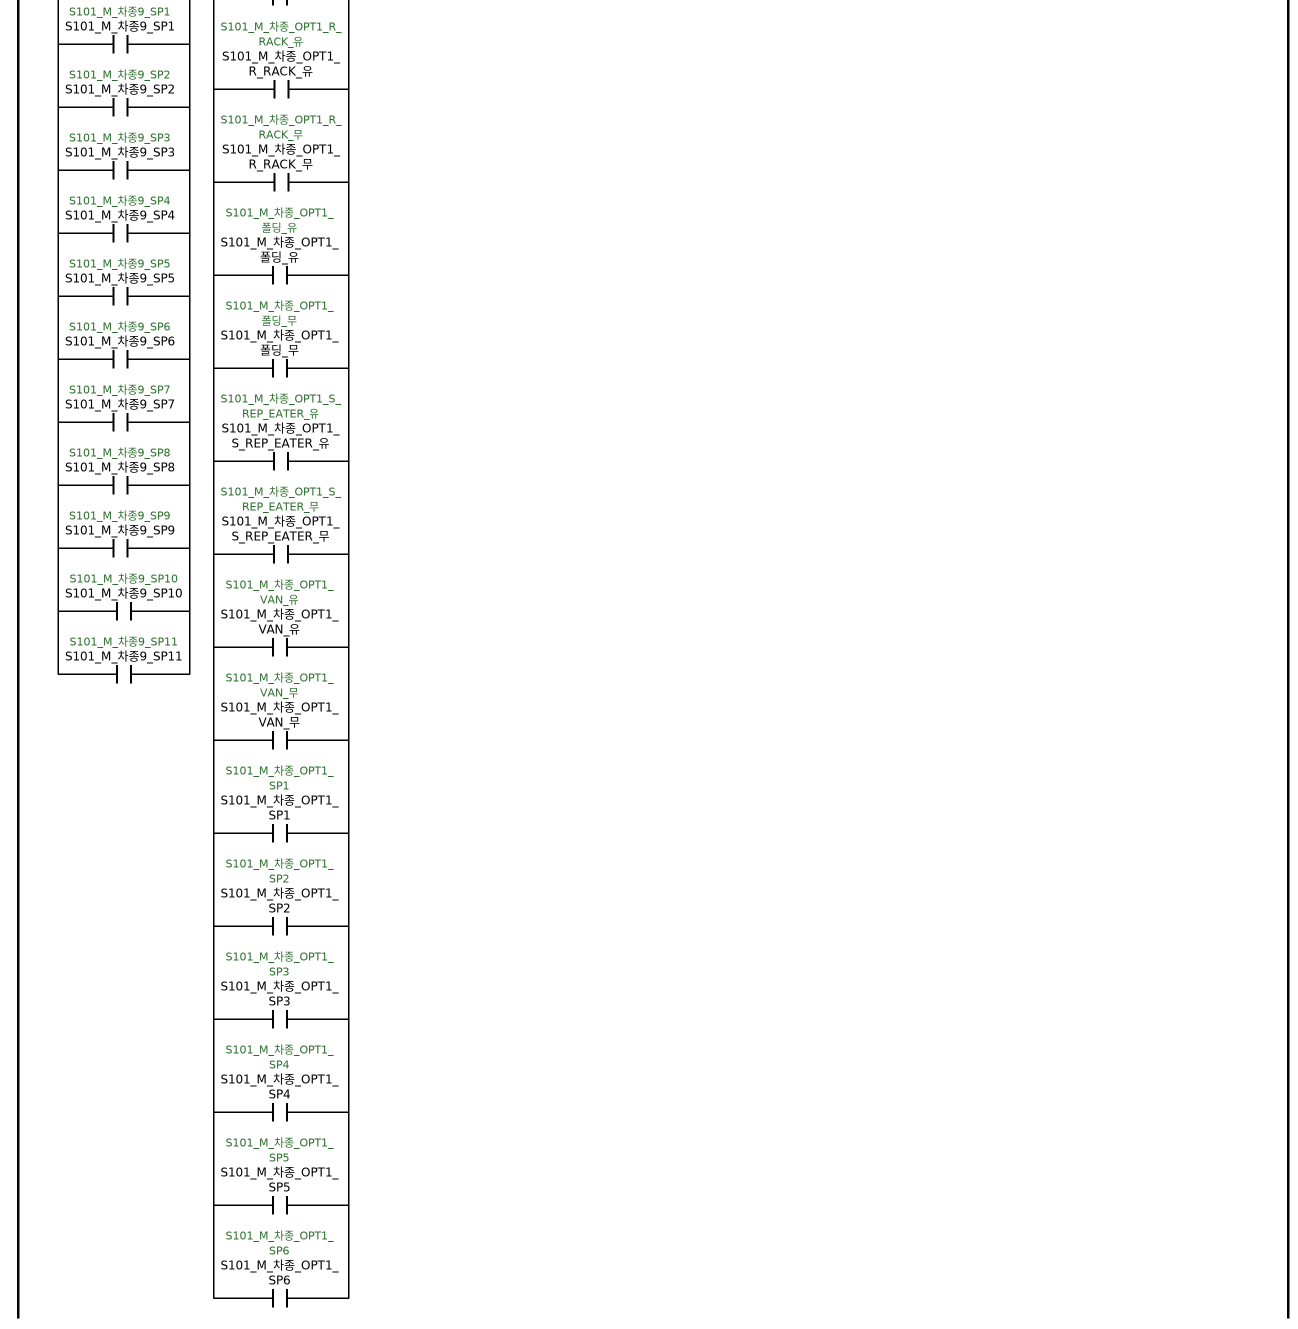
(* S101 차종 유 *)
(* Rung L72 *)
IF (S101_M_차종1_AX OR S101_M_차종1_B OR S101_M_차종1_C OR S101_M_차종1_D OR S101_M_차종1_E OR S101_M_차종1_F OR S101_M_차종1_G OR S101_M_차종1_H) AND (S101_M_차종2_3DR OR S101_M_차종2_4DR OR S101_M_차종2_5DR OR S101_M_차종2_WGN OR S101_M_차종2_SP1 OR S101_M_차종2_SP2) AND (S101_M_차종3_LHD OR S101_M_차종3_RHD) AND (S101_M_차종4_내수 OR S101_M_차종4_수출 OR S101_M_차종4_북미 OR S101_M_차종4_EEC OR S101_M_차종4_호주 OR S101_M_차종4_중동 OR S101_M_차종4_중국 OR S101_M_차종4_브라질 OR S101_M_차종4_SP1 OR S101_M_차종4_SP2 OR S101_M_차종4_러시아 OR S101_M_차종4_SP3 OR S101_M_차종4_SP4 OR S101_M_차종4_SP5 OR S101_M_차종4_SP6 OR S101_M_차종4_SP7) AND (S101_M_차종5_MT OR S101_M_차종5_AT OR S101_M_차종5_SP1) AND (S101_M_차종6_일반루프 OR S101_M_차종6_썬루프 OR S101_M_차종6_파노라마루프 OR S101_M_차종6_DSROOF OR S101_M_차종6_SP1) AND (S101_M_차종7_GSL OR S101_M_차종7_DSL OR S101_M_차종7_SP1 OR S101_M_차종7_SP2 OR S101_M_차종7_SP3 OR S101_M_차종7_SP4 OR S101_M_차종7_SP5 OR S101_M_차종7_SP6) AND (S101_M_차종8_2WD OR S101_M_차종8_4WD OR S101_M_차종8_SP1) AND (S101_M_차종9_MPI OR S101_M_차종9_T_GDI OR S101_M_차종9_SP1 OR S101_M_차종9_SP2 OR S101_M_차종9_SP3 OR S101_M_차종9_SP4 OR S101_M_차종9_SP5 OR S101_M_차종9_SP6 OR S101_M_차종9_SP7 OR S101_M_차종9_SP8 OR S101_M_차종9_SP9 OR S101_M_차종9_SP10 OR S101_M_차종9_SP11) AND (S101_M_차종_OPT1_슬라이딩_유 OR S101_M_차종_OPT1_슬라이딩_무 OR S101_M_차종_OPT1_R_RACK_유 OR S101_M_차종_OPT1_R_RACK_무 OR S101_M_차종_OPT1_폴딩_유 OR S101_M_차종_OPT1_폴딩_무 OR S101_M_차종_OPT1_S_REP_EATER_유 OR S101_M_차종_OPT1_S_REP_EATER_무 OR S101_M_차종_OPT1_VAN_유 OR S101_M_차종_OPT1_VAN_무 OR S101_M_차종_OPT1_SP1 OR S101_M_차종_OPT1_SP2 OR S101_M_차종_OPT1_SP3 OR S101_M_차종_OPT1_SP4 OR S101_M_차종_OPT1_SP5 OR S101_M_차종_OPT1_SP6) THEN
    _t2 := S101_M_SEQ <> 0;
END_IF;
S101_M_STN_차종_ON := _t2;

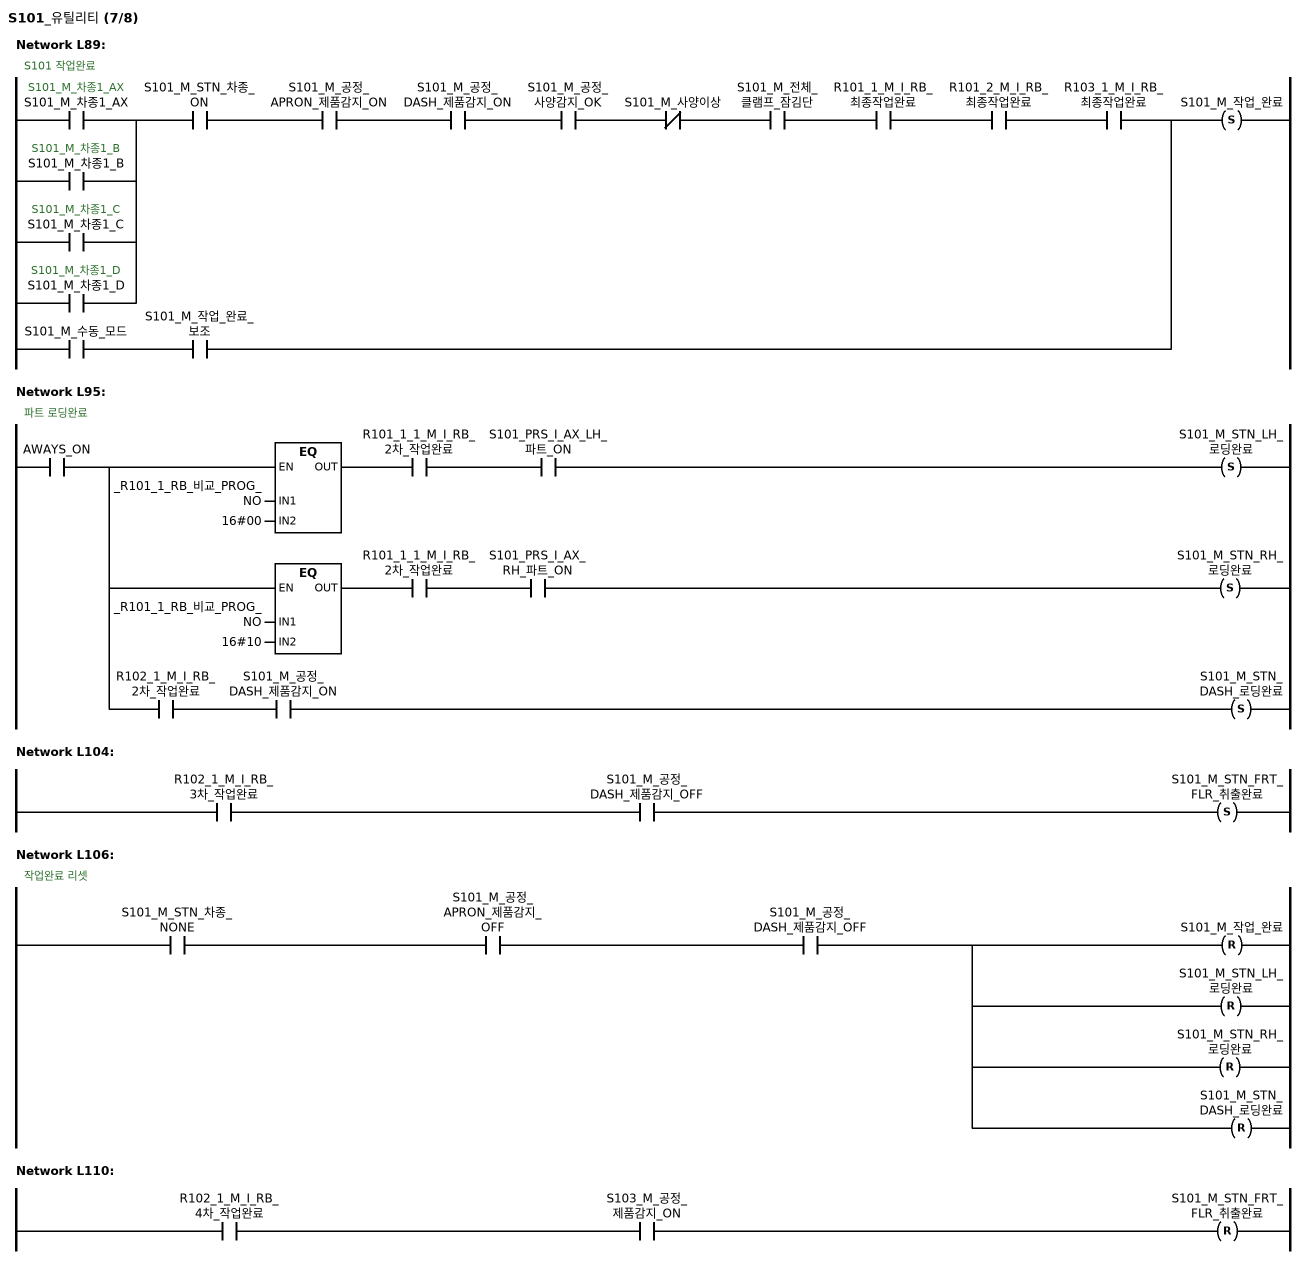
(* S101 작업완료 *)
(* Rung L89 *)
IF ((S101_M_차종1_AX OR S101_M_차종1_B OR S101_M_차종1_C OR S101_M_차종1_D) AND S101_M_STN_차종_ON AND S101_M_공정_APRON_제품감지_ON AND S101_M_공정_DASH_제품감지_ON AND S101_M_공정_사양감지_OK AND NOT S101_M_사양이상 AND S101_M_전체_클램프_잠김단 AND R101_1_M_I_RB_최종작업완료 AND R101_2_M_I_RB_최종작업완료 AND R103_1_M_I_RB_최종작업완료) OR (S101_M_수동_모드 AND S101_M_작업_완료_보조) THEN
    S101_M_작업_완료 := TRUE;
END_IF;
(* 파트 로딩완료 *)
(* Rung L95 *)
IF AWAYS_ON THEN _t3 := _R101_1_RB_비교_PROG_NO = 16#00; END_IF;
IF _t3 AND R101_1_1_M_I_RB_2차_작업완료 AND S101_PRS_I_AX_LH_파트_ON THEN S101_M_STN_LH_로딩완료 := TRUE; END_IF;
IF AWAYS_ON THEN _t4 := _R101_1_RB_비교_PROG_NO = 16#10; END_IF;
IF _t4 AND R101_1_1_M_I_RB_2차_작업완료 AND S101_PRS_I_AX_RH_파트_ON THEN S101_M_STN_RH_로딩완료 := TRUE; END_IF;
IF AWAYS_ON AND R102_1_M_I_RB_2차_작업완료 AND S101_M_공정_DASH_제품감지_ON THEN
    S101_M_STN_DASH_로딩완료 := TRUE;
END_IF;
(* Rung L104 *)
IF R102_1_M_I_RB_3차_작업완료 AND S101_M_공정_DASH_제품감지_OFF THEN S101_M_STN_FRT_FLR_취출완료 := TRUE; END_IF;
(* 작업완료 리셋 *)
(* Rung L106 *)
_p5 := S101_M_STN_차종_NONE AND S101_M_공정_APRON_제품감지_OFF AND S101_M_공정_DASH_제품감지_OFF;
IF _p5 THEN
    S101_M_작업_완료 := FALSE;
    S101_M_STN_LH_로딩완료 := FALSE;
    S101_M_STN_RH_로딩완료 := FALSE;
    S101_M_STN_DASH_로딩완료 := FALSE;
END_IF;
(* Rung L110 *)
IF R102_1_M_I_RB_4차_작업완료 AND S103_M_공정_제품감지_ON THEN S101_M_STN_FRT_FLR_취출완료 := FALSE; END_IF;

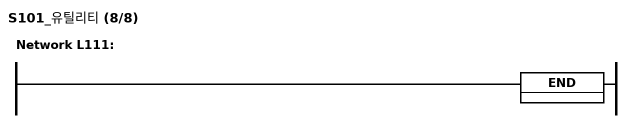
(* Rung L111 *)
END();
END_PROGRAM

PROGRAM S101_동작 (* task: 스캔 프로그램 *)
VAR
    ACC : INT;
    ACC2 : WORD;
    ACC3 : WORD;
    AX_3축_1_END : BOOL;
    AX_3축_1_전진단 : BOOL;
    AX_3축_1_후진단 : BOOL;
    AX_3축_2_전진단 : BOOL;
    AX_3축_2_후진단 : BOOL;
    AX_3축_3_전진단 : BOOL;
    AX_3축_3_후진단 : BOOL;
    DCEL : INT;
    DCEL2 : WORD;
    DCEL3 : WORD;
    HOME : BOOL;
    HOME_2 : BOOL;
    HOME_3 : BOOL;
    INST : TON;
    INST1 : TON;
    INST10 : TON;
    INST11 : TON;
    INST12 : TON;
    INST13 : TON;
    INST14 : TON;
    INST15 : TON;
    INST16 : TON;
    INST17 : TON;
    INST18 : TON;
    INST19 : TON;
    INST2 : TON;
    INST20 : TON;
    INST21 : TON;
    INST23 : TON;
    INST24 : TON;
    INST25 : TON;
    INST3 : TON;
    INST4 : TON;
    INST8 : TON;
    INST9 : TON;
    JOG_OFF : BOOL;
    JOG_OFF_2 : BOOL;
    JOG_OFF_3 : BOOL;
    JOG_ON : BOOL;
    JOG_ON_2 : BOOL;
    JOG_ON_3 : BOOL;
    limit : BOOL;
    ON : BOOL;
    OUT : DINT;
    OVERIDE : INT;
    OVERIDE2 : WORD;
    OVERIDE3 : WORD;
    POSION_1 : WORD;
    POSITION : DWORD;
    POSITION2 : DWORD;
    POSITION3 : DWORD;
    pp : BOOL;
    RST : BOOL;
    S103_핀클램프 : ACT_6_CYL;
    SRV3_START : TON;
    START : BOOL;
    START_2 : BOOL;
    START_3 : BOOL;
    sw1 : BOOL;
    SW10 : BOOL;
    SW10_2 : BOOL;
    SW10_3 : BOOL;
    SW11 : BOOL;
    SW11_2 : BOOL;
    SW11_3 : BOOL;
    SW12 : BOOL;
    SW12_2 : BOOL;
    SW12_3 : BOOL;
    sw1_2 : BOOL;
    sw1_3 : BOOL;
    sw2 : BOOL;
    sw2_2 : BOOL;
    sw2_3 : BOOL;
    sw3 : BOOL;
    SW4 : BOOL;
    SW4_2 : BOOL;
    SW4_3 : BOOL;
    SW5 : BOOL;
    SW6_2 : BOOL;
    SW6_3 : BOOL;
    SW7 : BOOL;
    SW7_2 : BOOL;
    SW7_3 : BOOL;
    TARGET_POSITION : DWORD;
    TARGET_POSITION2 : DWORD;
    TARGET_POSITION3 : DWORD;
    TEMP : BOOL;
    TEMP2 : BOOL;
    _3축2_전진단_보조1 : BOOL;
    _3축2_전진단_보조2 : BOOL;
    _3축2_후진단_보조1 : BOOL;
    _3축2_후진단_보조2 : BOOL;
    _3축3_전진단_보조1 : BOOL;
    _3축3_전진단_보조2 : BOOL;
    _3축3_후진단_보조1 : BOOL;
    _3축3_후진단_보조2 : BOOL;
    _3축_전진단_보조1 : BOOL;
    _3축_전진단_보조2 : BOOL;
    _3축_후진단_보조1 : BOOL;
    _3축_후진단_보조2 : BOOL;
    작업_COMP : TON;
    출력_속도값 : DWORD;
    출력_속도값2 : DWORD;
    출력_속도값3 : DWORD;
END_VAR
VAR_EXTERNAL
    AWAYS_ON : BOOL; (* AT %MW3.1 *)
    EGIS_EJS : BOOL;
    MCP_PBL_101_자동_운전 : BOOL; (* AT %MW87630.4 *) (* 입력 접점 04 *)
    MCP_PBL_운전준비_ON : BOOL; (* AT %MW87630.0 *) (* 입력 접점 00 *)
    MCP_SSP_101_수동_선택 : BOOL; (* AT %MW87630.2 *) (* 입력 접점 02 *)
    MCP_SSP_101_자동_선택 : BOOL; (* AT %MW87630.3 *) (* 입력 접점 03 *)
    R101_1_1_M_차종1_AX : BOOL; (* AT %MW10001.0 *) (* R101_1_1_M_차종1_AX *)
    S101_3축_1_ABSOLUTE : BOOL; (* AT %MW51002.8 *)
    S101_3축_1_ACCEL : WORD; (* AT %MW51009 *)
    S101_3축_1_COAST_정지 : BOOL; (* AT %MW51000.1 *)
    S101_3축_1_DECEL : WORD; (* AT %MW51010 *)
    S101_3축_1_ENALBLE1 : BOOL; (* AT %MW51000.0 *)
    S101_3축_1_ENALBLE2 : BOOL; (* AT %MW51000.3 *)
    S101_3축_1_FAULT : BOOL; (* AT %MW50000.3 *)
    S101_3축_1_HOME : BOOL; (* AT %MW51000.11 *)
    S101_3축_1_INTERME_정지 : BOOL; (* AT %MW51000.5 *)
    S101_3축_1_JOG_전진 : BOOL; (* AT %MW51000.8 *)
    S101_3축_1_JOG_후진 : BOOL; (* AT %MW51000.9 *)
    S101_3축_1_MDI_선택 : BOOL; (* AT %MW51001.15 *)
    S101_3축_1_MOVE_COMP : BOOL; (* AT %MW50000.10 *)
    S101_3축_1_OUT_VELOCITY1 : WORD; (* AT %MW51007 *)
    S101_3축_1_OUT_VELOCITY2 : WORD; (* AT %MW51008 *)
    S101_3축_1_OVERRIDE : WORD; (* AT %MW51004 *)
    S101_3축_1_PLC_CONTROL : BOOL; (* AT %MW51000.10 *)
    S101_3축_1_POSITION : DINT; (* AT %MD255 *)
    S101_3축_1_POSITION1 : WORD; (* AT %MW50005 *)
    S101_3축_1_POSITION2 : WORD; (* AT %MW50006 *)
    S101_3축_1_QUICK_정지 : BOOL; (* AT %MW51000.2 *)
    S101_3축_1_SOFT_LIMIT : BOOL; (* AT %MW51002.14 *)
    S101_3축_1_START1 : BOOL; (* AT %MW51000.4 *)
    S101_3축_1_START2 : BOOL; (* AT %MW51000.6 *)
    S101_3축_1_TARGET_POSITION : DINT; (* AT %MD280 *)
    S101_3축_1_TARGET_POSITION1 : WORD; (* AT %MW51005 *)
    S101_3축_1_TARGET_POSITION2 : WORD; (* AT %MW51006 *)
    S101_3축_1_TRACK_모드 : BOOL; (* AT %MW51002.0 *)
    S101_3축_1_운전준비1 : BOOL; (* AT %MW50000.0 *)
    S101_3축_1_운전준비2 : BOOL; (* AT %MW50000.1 *)
    S101_3축_1_운전준비_COMP : BOOL; (* AT %MW50000.2 *)
    S101_3축_1_이상_리셋 : BOOL; (* AT %MW51000.7 *)
    S101_3축_2_ABSOLUTE : BOOL; (* AT %MW51102.8 *)
    S101_3축_2_ACCEL : WORD; (* AT %MW51109 *)
    S101_3축_2_COAST_정지 : BOOL; (* AT %MW51100.1 *)
    S101_3축_2_DECEL : WORD; (* AT %MW51110 *)
    S101_3축_2_ENALBLE1 : BOOL; (* AT %MW51100.0 *)
    S101_3축_2_ENALBLE2 : BOOL; (* AT %MW51100.3 *)
    S101_3축_2_FAULT : BOOL; (* AT %MW50100.3 *)
    S101_3축_2_HOME : BOOL; (* AT %MW51100.11 *)
    S101_3축_2_INTERME_정지 : BOOL; (* AT %MW51100.5 *)
    S101_3축_2_JOG_전진 : BOOL; (* AT %MW51100.8 *)
    S101_3축_2_JOG_후진 : BOOL; (* AT %MW51100.9 *)
    S101_3축_2_MDI_선택 : BOOL; (* AT %MW51101.15 *)
    S101_3축_2_MOVE_COMP : BOOL; (* AT %MW50100.10 *)
    S101_3축_2_OUT_VELOCITY1 : WORD; (* AT %MW51107 *)
    S101_3축_2_OUT_VELOCITY2 : WORD; (* AT %MW51108 *)
    S101_3축_2_OVERRIDE : WORD; (* AT %MW51104 *)
    S101_3축_2_PLC_CONTROL : BOOL; (* AT %MW51100.10 *)
    S101_3축_2_POSITION : DINT; (* AT %MD260 *)
    S101_3축_2_POSITION1 : WORD; (* AT %MW50105 *)
    S101_3축_2_POSITION2 : WORD; (* AT %MW50106 *)
    S101_3축_2_QUICK_정지 : BOOL; (* AT %MW51100.2 *)
    S101_3축_2_SOFT_LIMIT : BOOL; (* AT %MW51102.14 *)
    S101_3축_2_START1 : BOOL; (* AT %MW51100.4 *)
    S101_3축_2_START2 : BOOL; (* AT %MW51100.6 *)
    S101_3축_2_TARGET_POSITION : DINT; (* AT %MD285 *)
    S101_3축_2_TARGET_POSITION1 : WORD; (* AT %MW51105 *)
    S101_3축_2_TARGET_POSITION2 : WORD; (* AT %MW51106 *)
    S101_3축_2_TRACK_모드 : BOOL; (* AT %MW51102.0 *)
    S101_3축_2_운전준비1 : BOOL; (* AT %MW50100.0 *)
    S101_3축_2_운전준비2 : BOOL; (* AT %MW50100.1 *)
    S101_3축_2_운전준비_COMP : BOOL; (* AT %MW50100.2 *)
    S101_3축_2_이상_리셋 : BOOL; (* AT %MW51100.7 *)
    S101_3축_3_ABSOLUTE : BOOL; (* AT %MW51202.8 *)
    S101_3축_3_ACCEL : WORD; (* AT %MW51209 *)
    S101_3축_3_COAST_정지 : BOOL; (* AT %MW51200.1 *)
    S101_3축_3_DECEL : WORD; (* AT %MW51210 *)
    S101_3축_3_ENALBLE1 : BOOL; (* AT %MW51200.0 *)
    S101_3축_3_ENALBLE2 : BOOL; (* AT %MW51200.3 *)
    S101_3축_3_FAULT : BOOL; (* AT %MW50200.3 *)
    S101_3축_3_HOME : BOOL; (* AT %MW51200.11 *)
    S101_3축_3_INTERME_정지 : BOOL; (* AT %MW51200.5 *)
    S101_3축_3_JOG_전진 : BOOL; (* AT %MW51200.8 *)
    S101_3축_3_JOG_후진 : BOOL; (* AT %MW51200.9 *)
    S101_3축_3_MDI_선택 : BOOL; (* AT %MW51201.15 *)
    S101_3축_3_MOVE_COMP : BOOL; (* AT %MW50200.10 *)
    S101_3축_3_OUT_VELOCITY1 : WORD; (* AT %MW51207 *)
    S101_3축_3_OUT_VELOCITY2 : WORD; (* AT %MW51208 *)
    S101_3축_3_OVERRIDE : WORD; (* AT %MW51204 *)
    S101_3축_3_PLC_CONTROL : BOOL; (* AT %MW51200.10 *)
    S101_3축_3_POSITION : DINT; (* AT %MD265 *)
    S101_3축_3_POSITION1 : WORD; (* AT %MW50205 *)
    S101_3축_3_POSITION2 : WORD; (* AT %MW50206 *)
    S101_3축_3_QUICK_정지 : BOOL; (* AT %MW51200.2 *)
    S101_3축_3_SOFT_LIMIT : BOOL; (* AT %MW51202.14 *)
    S101_3축_3_TARGET_POSITION : DINT; (* AT %MD290 *)
    S101_3축_3_TARGET_POSITION1 : WORD; (* AT %MW51205 *)
    S101_3축_3_TARGET_POSITION2 : WORD; (* AT %MW51206 *)
    S101_3축_3_TRACK_모드 : BOOL; (* AT %MW51202.0 *)
    S101_3축_3_운전준비1 : BOOL; (* AT %MW50200.0 *)
    S101_3축_3_운전준비2 : BOOL; (* AT %MW50200.1 *)
    S101_3축_3_운전준비_COMP : BOOL; (* AT %MW50200.2 *)
    S101_3축_3_이상_리셋 : BOOL; (* AT %MW51200.7 *)
    S101_6_10_PLC_BOX_CP_TRIP : BOOL; (* AT %MW86102.15 *) (* 입력 접점 15 *)
    S101_AX_래치 : ACT_6_CYL;
    S101_DASH_클램프 : ACT_6_CYL;
    S101_HOME : BOOL; (* AT %MW1048.0 *)
    S101_JOG_OFF : BOOL; (* AT %MW1048.5 *)
    S101_JOG_ON : BOOL; (* AT %MW1048.4 *)
    S101_MCR_비상정지1 : BOOL; (* AT %MW95207.0 *) (* 출력 접점 00 *)
    S101_MCR_비상정지2 : BOOL; (* AT %MW95207.1 *) (* 출력 접점 01 *)
    S101_MCR_비상정지3 : BOOL; (* AT %MW95207.2 *) (* 출력 접점 02 *)
    S101_M_3_축1_전진_보조 : BOOL; (* AT %MW1102.1 *)
    S101_M_3_축1_전진단 : BOOL; (* AT %MW1102.3 *)
    S101_M_3_축1_조건 : BOOL; (* AT %MW1102.0 *)
    S101_M_3_축1_후진_보조 : BOOL; (* AT %MW1102.2 *)
    S101_M_3_축1_후진단 : BOOL; (* AT %MW1102.4 *)
    S101_M_3_축2_전진_보조 : BOOL; (* AT %MW1103.1 *)
    S101_M_3_축2_전진단 : BOOL; (* AT %MW1103.3 *)
    S101_M_3_축2_조건 : BOOL; (* AT %MW1103.0 *)
    S101_M_3_축2_후진_보조 : BOOL; (* AT %MW1103.2 *)
    S101_M_3_축2_후진단 : BOOL; (* AT %MW1103.4 *)
    S101_M_3_축3_전진_보조 : BOOL; (* AT %MW1104.1 *)
    S101_M_3_축3_전진단 : BOOL; (* AT %MW1104.3 *)
    S101_M_3_축3_조건 : BOOL; (* AT %MW1104.0 *)
    S101_M_3_축3_후진_보조 : BOOL; (* AT %MW1104.2 *)
    S101_M_3_축3_후진단 : BOOL; (* AT %MW1104.4 *)
    S101_M_ACT_선택_1 : BOOL; (* AT %MW1040.0 *)
    S101_M_ACT_선택_2 : BOOL; (* AT %MW1040.1 *)
    S101_M_ACT_선택_3 : BOOL; (* AT %MW1040.2 *)
    S101_M_ACT_선택_4 : BOOL; (* AT %MW1040.3 *)
    S101_M_ACT_선택_5 : BOOL; (* AT %MW1040.4 *)
    S101_M_ACT_선택_6 : BOOL; (* AT %MW1040.5 *)
    S101_M_ACT_선택_7 : BOOL; (* AT %MW1040.6 *)
    S101_M_AX_래치_전진_LAMP : WORD; (* AT %MW11100 *)
    S101_M_AX_래치_전진_LS_이상 : BOOL; (* AT %MW1100.5 *)
    S101_M_AX_래치_전진_보조 : BOOL; (* AT %MW1100.1 *)
    S101_M_AX_래치_전진단 : BOOL; (* AT %MW1100.3 *)
    S101_M_AX_래치_조건 : BOOL; (* AT %MW1100.0 *)
    S101_M_AX_래치_후진_LAMP : WORD; (* AT %MW11101 *)
    S101_M_AX_래치_후진_LS_이상 : BOOL; (* AT %MW1100.6 *)
    S101_M_AX_래치_후진_보조 : BOOL; (* AT %MW1100.2 *)
    S101_M_AX_래치_후진단 : BOOL; (* AT %MW1100.4 *)
    S101_M_DASH_클램프_전진_LAMP : WORD; (* AT %MW11104 *)
    S101_M_DASH_클램프_전진_LS_이상 : BOOL; (* AT %MW1105.5 *)
    S101_M_DASH_클램프_전진_보조 : BOOL; (* AT %MW1105.1 *)
    S101_M_DASH_클램프_전진단 : BOOL; (* AT %MW1105.3 *)
    S101_M_DASH_클램프_조건 : BOOL; (* AT %MW1105.0 *)
    S101_M_DASH_클램프_후진_LAMP : WORD; (* AT %MW11105 *)
    S101_M_DASH_클램프_후진_LS_이상 : BOOL; (* AT %MW1105.6 *)
    S101_M_DASH_클램프_후진_보조 : BOOL; (* AT %MW1105.2 *)
    S101_M_DASH_클램프_후진단 : BOOL; (* AT %MW1105.4 *)
    S101_M_SHIFT_전진_LAMP : WORD; (* AT %MW11102 *)
    S101_M_SHIFT_전진_LS_이상 : BOOL; (* AT %MW1101.5 *)
    S101_M_SHIFT_전진_보조 : BOOL; (* AT %MW1101.1 *)
    S101_M_SHIFT_전진단 : BOOL; (* AT %MW1101.3 *)
    S101_M_SHIFT_조건 : BOOL; (* AT %MW1101.0 *)
    S101_M_SHIFT_후진_LAMP : WORD; (* AT %MW11103 *)
    S101_M_SHIFT_후진_LS_이상 : BOOL; (* AT %MW1101.6 *)
    S101_M_SHIFT_후진_보조 : BOOL; (* AT %MW1101.2 *)
    S101_M_SHIFT_후진단 : BOOL; (* AT %MW1101.4 *)
    S101_M_공정_APRON_제품감지_OFF : BOOL; (* AT %MW1001.4 *)
    S101_M_공정_APRON_제품감지_ON : BOOL; (* AT %MW1001.3 *)
    S101_M_공정_DASH_제품감지_OFF : BOOL; (* AT %MW1001.6 *)
    S101_M_공정_DASH_제품감지_ON : BOOL; (* AT %MW1001.5 *)
    S101_M_공정_HOME_POSI : BOOL; (* AT %MW1004.0 *)
    S101_M_공정_간섭무 : BOOL; (* AT %MW1004.1 *)
    S101_M_수동_모드 : BOOL; (* AT %MW1000.3 *)
    S101_M_운전준비_ON : BOOL; (* AT %MW1000.0 *)
    S101_M_자동_START : BOOL; (* AT %MW1000.5 *)
    S101_M_자동_모드 : BOOL; (* AT %MW1000.1 *)
    S101_M_자동_운전중 : BOOL; (* AT %MW1000.4 *)
    S101_M_작업_완료 : BOOL; (* AT %MW1001.0 *)
    S101_M_총괄_CP_이상 : BOOL; (* AT %MW1009.7 *)
    S101_M_총괄_CT_이상 : BOOL; (* AT %MW1010.4 *)
    S101_M_총괄_EOCR_이상 : BOOL; (* AT %MW1009.8 *)
    S101_M_총괄_INV_이상 : BOOL; (* AT %MW1009.9 *)
    S101_M_총괄_LS_이상 : BOOL; (* AT %MW1009.15 *)
    S101_M_총괄_MATCH_이상 : BOOL; (* AT %MW1010.0 *)
    S101_M_총괄_MC_이상 : BOOL; (* AT %MW1009.13 *)
    S101_M_총괄_NFB_이상 : BOOL; (* AT %MW1009.11 *)
    S101_M_총괄_ROBOT_이상 : BOOL; (* AT %MW1010.1 *)
    S101_M_총괄_SAFETY_이상 : BOOL; (* AT %MW1009.2 *)
    S101_M_총괄_공기압_이상 : BOOL; (* AT %MW1009.3 *)
    S101_M_총괄_사양_이상 : BOOL; (* AT %MW1009.6 *)
    S101_M_총괄_오버런_이상 : BOOL; (* AT %MW1009.12 *)
    S101_M_총괄_용점타점수_이상 : BOOL; (* AT %MW1010.2 *)
    S101_M_총괄_이상 : BOOL; (* AT %MW1009.0 *)
    S101_M_총괄_제품감지_이상 : BOOL; (* AT %MW1009.4 *)
    S101_M_총괄_차종_이상 : BOOL; (* AT %MW1009.5 *)
    S101_M_총괄_통신_이상 : BOOL; (* AT %MW1009.14 *)
    S101_M_핀클램프_전진_LAMP : WORD; (* AT %MW11106 *)
    S101_M_핀클램프_전진_LS_이상 : BOOL; (* AT %MW1106.5 *)
    S101_M_핀클램프_전진_보조 : BOOL; (* AT %MW1106.1 *)
    S101_M_핀클램프_전진단 : BOOL; (* AT %MW1106.3 *)
    S101_M_핀클램프_조건 : BOOL; (* AT %MW1106.0 *)
    S101_M_핀클램프_후진_LAMP : WORD; (* AT %MW11107 *)
    S101_M_핀클램프_후진_LS_이상 : BOOL; (* AT %MW1106.6 *)
    S101_M_핀클램프_후진_보조 : BOOL; (* AT %MW1106.2 *)
    S101_M_핀클램프_후진단 : BOOL; (* AT %MW1106.4 *)
    S101_PRS_AX_DASH_클램프_전진 : BOOL; (* AT %MW86100.13 *) (* 입력 접점 13 *)
    S101_PRS_AX_DASH_클램프_후진 : BOOL; (* AT %MW86100.12 *) (* 입력 접점 12 *)
    S101_PRS_AX_핀클램프_전진단1 : BOOL; (* AT %MW86101.0 *)
    S101_PRS_AX_핀클램프_전진단2 : BOOL; (* AT %MW86101.2 *)
    S101_PRS_AX_핀클램프_전진단3 : BOOL; (* AT %MW86101.4 *)
    S101_PRS_AX_핀클램프_전진단4 : BOOL; (* AT %MW86101.6 *)
    S101_PRS_AX_핀클램프_후진단1 : BOOL; (* AT %MW86101.1 *)
    S101_PRS_AX_핀클램프_후진단2 : BOOL; (* AT %MW86101.3 *)
    S101_PRS_AX_핀클램프_후진단3 : BOOL; (* AT %MW86101.5 *)
    S101_PRS_AX_핀클램프_후진단4 : BOOL; (* AT %MW86101.7 *)
    S101_RS_AX_SFT_전진1 : BOOL; (* AT %MW86100.8 *) (* 입력 접점 08 *)
    S101_RS_AX_SFT_전진2 : BOOL; (* AT %MW86100.10 *) (* 입력 접점 10 *)
    S101_RS_AX_SFT_후진1 : BOOL; (* AT %MW86100.9 *) (* 입력 접점 09 *)
    S101_RS_AX_SFT_후진2 : BOOL; (* AT %MW86100.11 *) (* 입력 접점 11 *)
    S101_RS_AX_래치_전진1 : BOOL; (* AT %MW86100.0 *) (* 입력 접점 00 *)
    S101_RS_AX_래치_전진2 : BOOL; (* AT %MW86100.2 *) (* 입력 접점 02 *)
    S101_RS_AX_래치_후진1 : BOOL; (* AT %MW86100.1 *) (* 입력 접점 01 *)
    S101_RS_AX_래치_후진2 : BOOL; (* AT %MW86100.3 *) (* 입력 접점 03 *)
    S101_SHIFT : ACT_6_CYL;
    S101_SOL_AX_DASH_클램프_전진 : BOOL; (* AT %MW96103.4 *) (* 출력 접점 04 *)
    S101_SOL_AX_DASH_클램프_후진 : BOOL; (* AT %MW96103.5 *) (* 출력 접점 05 *)
    S101_SOL_AX_SHIFT_전진 : BOOL; (* AT %MW96103.2 *) (* 출력 접점 02 *)
    S101_SOL_AX_SHIFT_후진 : BOOL; (* AT %MW96103.3 *) (* 출력 접점 03 *)
    S101_SOL_AX_래치_전진 : BOOL; (* AT %MW96103.0 *) (* 출력 접점 00 *)
    S101_SOL_AX_래치_후진 : BOOL; (* AT %MW96103.1 *) (* 출력 접점 01 *)
    S101_SOL_AX_핀클램프_전진출력 : BOOL; (* AT %MW96103.6 *)
    S101_SOL_AX_핀클램프_후진출력 : BOOL; (* AT %MW96103.7 *)
    S101_공기압_AIR_CHECK : BOOL; (* AT %MW86102.14 *) (* 입력 접점 14 *)
    S101_운전준비 : TON;
    S101_전진_ON : BOOL; (* AT %MW1048.1 *)
    S101_후진_ON : BOOL; (* AT %MW1048.2 *)
    S102_DASH_클램프 : ACT_6_CYL;
    S102_SHIFT : ACT_6_CYL;
    S103_DASH_클램프 : ACT_6_CYL;
    SW6 : BOOL;
    T101_자동 : TON;
    T102_자동 : TON;
    TEST1 : BOOL;
    전체_M_이상_리셋 : BOOL; (* AT %MW308.2 *) (* 전체 M 이상 리셋 *)
    전체_라인_M_총괄_SAFETY_이상 : BOOL; (* AT %MW300.2 *)
    전체_라인_M_총괄_공기압_이상 : BOOL; (* AT %MW300.3 *)
    전체_라인_M_총괄_비상정지_이상 : BOOL; (* AT %MW300.1 *)
    전체_라인_M_총괄_이상 : BOOL; (* AT %MW300.0 *)
END_VAR
VAR
    _t1 : BOOL;
    _t2 : BOOL;
    _t3 : BOOL;
END_VAR

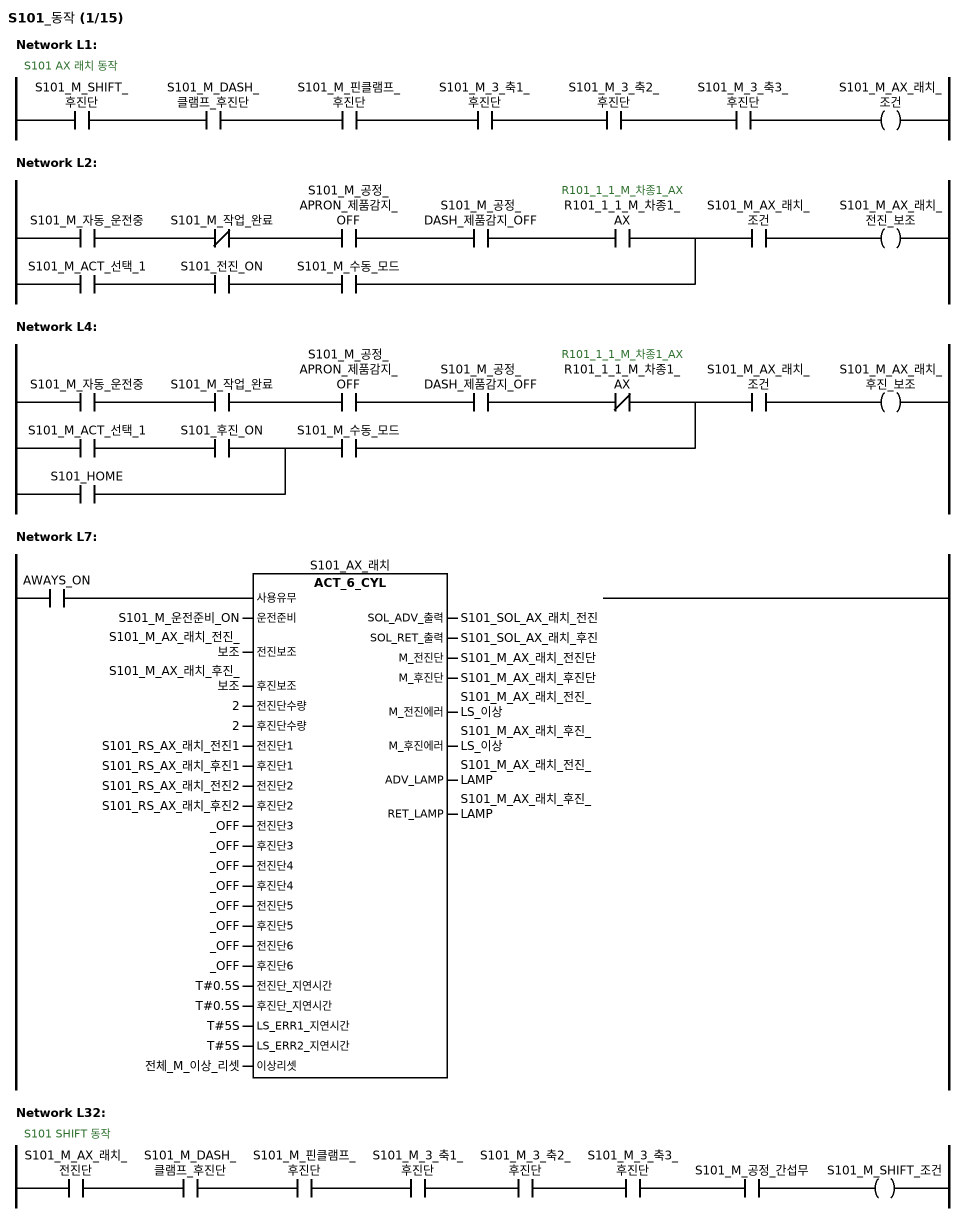
(* S101 AX 래치 동작 *)
(* Rung L1 *)
S101_M_AX_래치_조건 := S101_M_SHIFT_후진단 AND S101_M_DASH_클램프_후진단 AND S101_M_핀클램프_후진단 AND S101_M_3_축1_후진단 AND S101_M_3_축2_후진단 AND S101_M_3_축3_후진단;
(* Rung L2 *)
S101_M_AX_래치_전진_보조 := ((S101_M_자동_운전중 AND NOT S101_M_작업_완료 AND S101_M_공정_APRON_제품감지_OFF AND S101_M_공정_DASH_제품감지_OFF AND R101_1_1_M_차종1_AX) OR (S101_M_ACT_선택_1 AND S101_전진_ON AND S101_M_수동_모드)) AND S101_M_AX_래치_조건;
(* Rung L4 *)
S101_M_AX_래치_후진_보조 := ((S101_M_자동_운전중 AND S101_M_작업_완료 AND S101_M_공정_APRON_제품감지_OFF AND S101_M_공정_DASH_제품감지_OFF AND NOT R101_1_1_M_차종1_AX) OR (((S101_M_ACT_선택_1 AND S101_후진_ON) OR S101_HOME) AND S101_M_수동_모드)) AND S101_M_AX_래치_조건;
(* Rung L7 *)
S101_AX_래치(사용유무 := AWAYS_ON, 운전준비 := S101_M_운전준비_ON, 전진보조 := S101_M_AX_래치_전진_보조, 후진보조 := S101_M_AX_래치_후진_보조, 전진단수량 := 2, 후진단수량 := 2, 전진단1 := S101_RS_AX_래치_전진1, 후진단1 := S101_RS_AX_래치_후진1, 전진단2 := S101_RS_AX_래치_전진2, 후진단2 := S101_RS_AX_래치_후진2, 전진단3 := _OFF, 후진단3 := _OFF, 전진단4 := _OFF, 후진단4 := _OFF, 전진단5 := _OFF, 후진단5 := _OFF, 전진단6 := _OFF, 후진단6 := _OFF, 전진단_지연시간 := T#0.5S, 후진단_지연시간 := T#0.5S, LS_ERR1_지연시간 := T#5S, LS_ERR2_지연시간 := T#5S, 이상리셋 := 전체_M_이상_리셋, SOL_ADV_출력 => S101_SOL_AX_래치_전진, SOL_RET_출력 => S101_SOL_AX_래치_후진, M_전진단 => S101_M_AX_래치_전진단, M_후진단 => S101_M_AX_래치_후진단, M_전진에러 => S101_M_AX_래치_전진_LS_이상, M_후진에러 => S101_M_AX_래치_후진_LS_이상, ADV_LAMP => S101_M_AX_래치_전진_LAMP, RET_LAMP => S101_M_AX_래치_후진_LAMP);
(* S101 SHIFT 동작 *)
(* Rung L32 *)
S101_M_SHIFT_조건 := S101_M_AX_래치_전진단 AND S101_M_DASH_클램프_후진단 AND S101_M_핀클램프_후진단 AND S101_M_3_축1_후진단 AND S101_M_3_축2_후진단 AND S101_M_3_축3_후진단 AND S101_M_공정_간섭무;

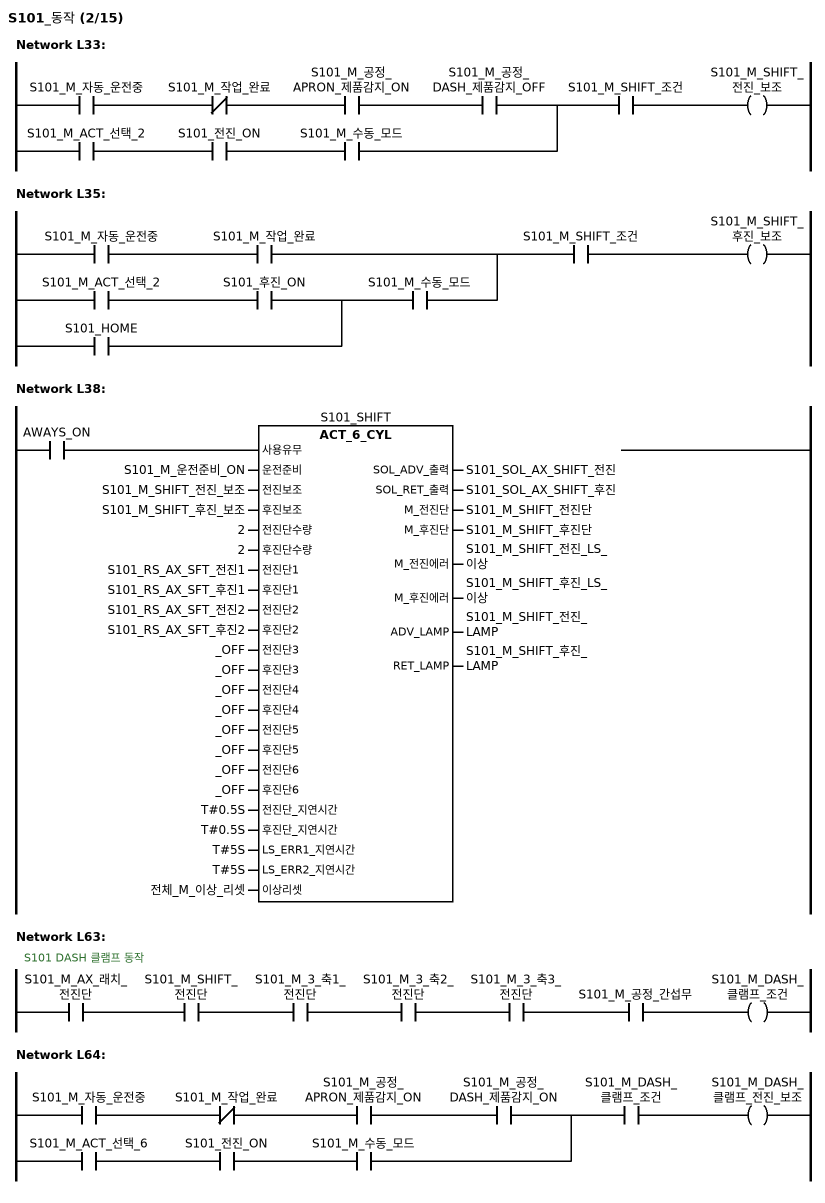
(* Rung L33 *)
S101_M_SHIFT_전진_보조 := ((S101_M_자동_운전중 AND NOT S101_M_작업_완료 AND S101_M_공정_APRON_제품감지_ON AND S101_M_공정_DASH_제품감지_OFF) OR (S101_M_ACT_선택_2 AND S101_전진_ON AND S101_M_수동_모드)) AND S101_M_SHIFT_조건;
(* Rung L35 *)
S101_M_SHIFT_후진_보조 := ((S101_M_자동_운전중 AND S101_M_작업_완료) OR (((S101_M_ACT_선택_2 AND S101_후진_ON) OR S101_HOME) AND S101_M_수동_모드)) AND S101_M_SHIFT_조건;
(* Rung L38 *)
S101_SHIFT(사용유무 := AWAYS_ON, 운전준비 := S101_M_운전준비_ON, 전진보조 := S101_M_SHIFT_전진_보조, 후진보조 := S101_M_SHIFT_후진_보조, 전진단수량 := 2, 후진단수량 := 2, 전진단1 := S101_RS_AX_SFT_전진1, 후진단1 := S101_RS_AX_SFT_후진1, 전진단2 := S101_RS_AX_SFT_전진2, 후진단2 := S101_RS_AX_SFT_후진2, 전진단3 := _OFF, 후진단3 := _OFF, 전진단4 := _OFF, 후진단4 := _OFF, 전진단5 := _OFF, 후진단5 := _OFF, 전진단6 := _OFF, 후진단6 := _OFF, 전진단_지연시간 := T#0.5S, 후진단_지연시간 := T#0.5S, LS_ERR1_지연시간 := T#5S, LS_ERR2_지연시간 := T#5S, 이상리셋 := 전체_M_이상_리셋, SOL_ADV_출력 => S101_SOL_AX_SHIFT_전진, SOL_RET_출력 => S101_SOL_AX_SHIFT_후진, M_전진단 => S101_M_SHIFT_전진단, M_후진단 => S101_M_SHIFT_후진단, M_전진에러 => S101_M_SHIFT_전진_LS_이상, M_후진에러 => S101_M_SHIFT_후진_LS_이상, ADV_LAMP => S101_M_SHIFT_전진_LAMP, RET_LAMP => S101_M_SHIFT_후진_LAMP);
(* S101 DASH 클램프 동작 *)
(* Rung L63 *)
S101_M_DASH_클램프_조건 := S101_M_AX_래치_전진단 AND S101_M_SHIFT_전진단 AND S101_M_3_축1_전진단 AND S101_M_3_축2_전진단 AND S101_M_3_축3_전진단 AND S101_M_공정_간섭무;
(* Rung L64 *)
S101_M_DASH_클램프_전진_보조 := ((S101_M_자동_운전중 AND NOT S101_M_작업_완료 AND S101_M_공정_APRON_제품감지_ON AND S101_M_공정_DASH_제품감지_ON) OR (S101_M_ACT_선택_6 AND S101_전진_ON AND S101_M_수동_모드)) AND S101_M_DASH_클램프_조건;

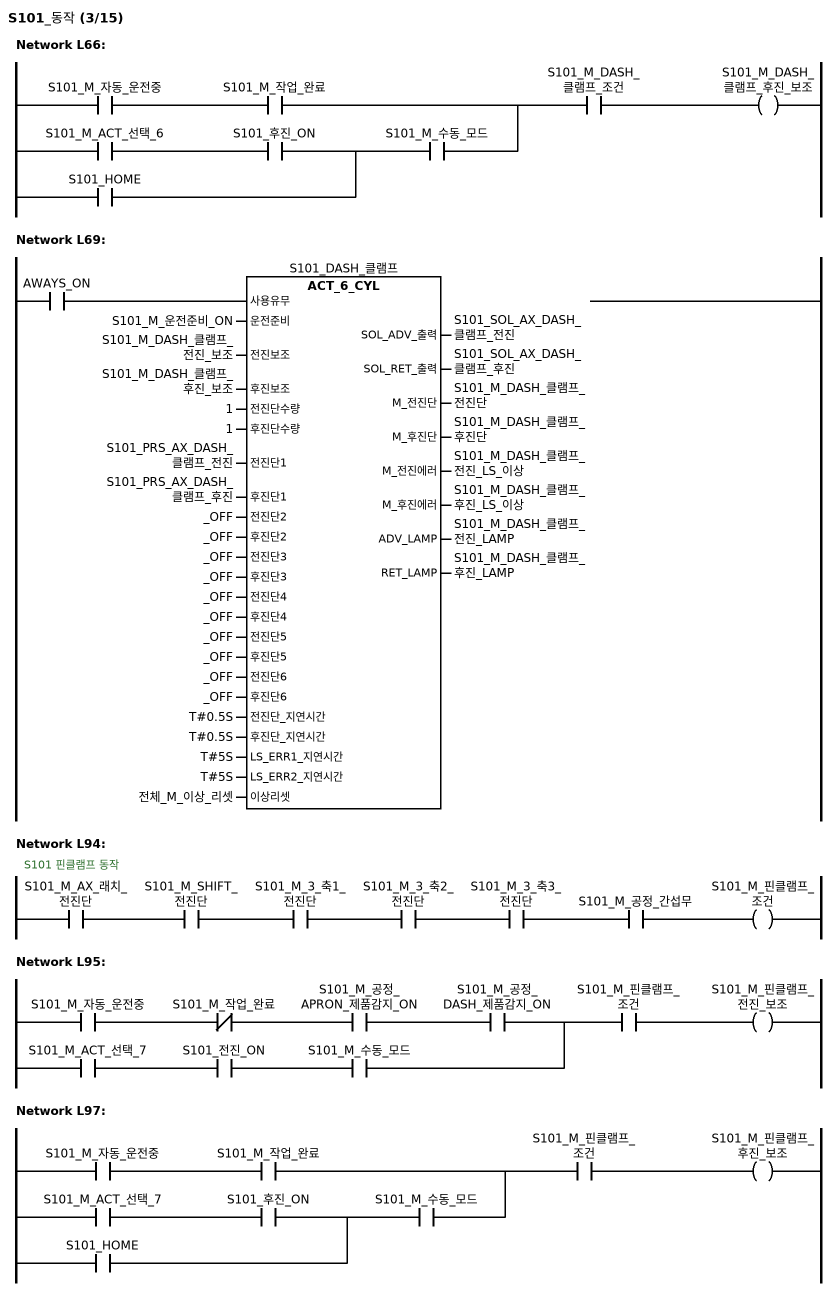
(* Rung L66 *)
S101_M_DASH_클램프_후진_보조 := ((S101_M_자동_운전중 AND S101_M_작업_완료) OR (((S101_M_ACT_선택_6 AND S101_후진_ON) OR S101_HOME) AND S101_M_수동_모드)) AND S101_M_DASH_클램프_조건;
(* Rung L69 *)
S101_DASH_클램프(사용유무 := AWAYS_ON, 운전준비 := S101_M_운전준비_ON, 전진보조 := S101_M_DASH_클램프_전진_보조, 후진보조 := S101_M_DASH_클램프_후진_보조, 전진단수량 := 1, 후진단수량 := 1, 전진단1 := S101_PRS_AX_DASH_클램프_전진, 후진단1 := S101_PRS_AX_DASH_클램프_후진, 전진단2 := _OFF, 후진단2 := _OFF, 전진단3 := _OFF, 후진단3 := _OFF, 전진단4 := _OFF, 후진단4 := _OFF, 전진단5 := _OFF, 후진단5 := _OFF, 전진단6 := _OFF, 후진단6 := _OFF, 전진단_지연시간 := T#0.5S, 후진단_지연시간 := T#0.5S, LS_ERR1_지연시간 := T#5S, LS_ERR2_지연시간 := T#5S, 이상리셋 := 전체_M_이상_리셋, SOL_ADV_출력 => S101_SOL_AX_DASH_클램프_전진, SOL_RET_출력 => S101_SOL_AX_DASH_클램프_후진, M_전진단 => S101_M_DASH_클램프_전진단, M_후진단 => S101_M_DASH_클램프_후진단, M_전진에러 => S101_M_DASH_클램프_전진_LS_이상, M_후진에러 => S101_M_DASH_클램프_후진_LS_이상, ADV_LAMP => S101_M_DASH_클램프_전진_LAMP, RET_LAMP => S101_M_DASH_클램프_후진_LAMP);
(* S101 핀클램프 동작 *)
(* Rung L94 *)
S101_M_핀클램프_조건 := S101_M_AX_래치_전진단 AND S101_M_SHIFT_전진단 AND S101_M_3_축1_전진단 AND S101_M_3_축2_전진단 AND S101_M_3_축3_전진단 AND S101_M_공정_간섭무;
(* Rung L95 *)
S101_M_핀클램프_전진_보조 := ((S101_M_자동_운전중 AND NOT S101_M_작업_완료 AND S101_M_공정_APRON_제품감지_ON AND S101_M_공정_DASH_제품감지_ON) OR (S101_M_ACT_선택_7 AND S101_전진_ON AND S101_M_수동_모드)) AND S101_M_핀클램프_조건;
(* Rung L97 *)
S101_M_핀클램프_후진_보조 := ((S101_M_자동_운전중 AND S101_M_작업_완료) OR (((S101_M_ACT_선택_7 AND S101_후진_ON) OR S101_HOME) AND S101_M_수동_모드)) AND S101_M_핀클램프_조건;

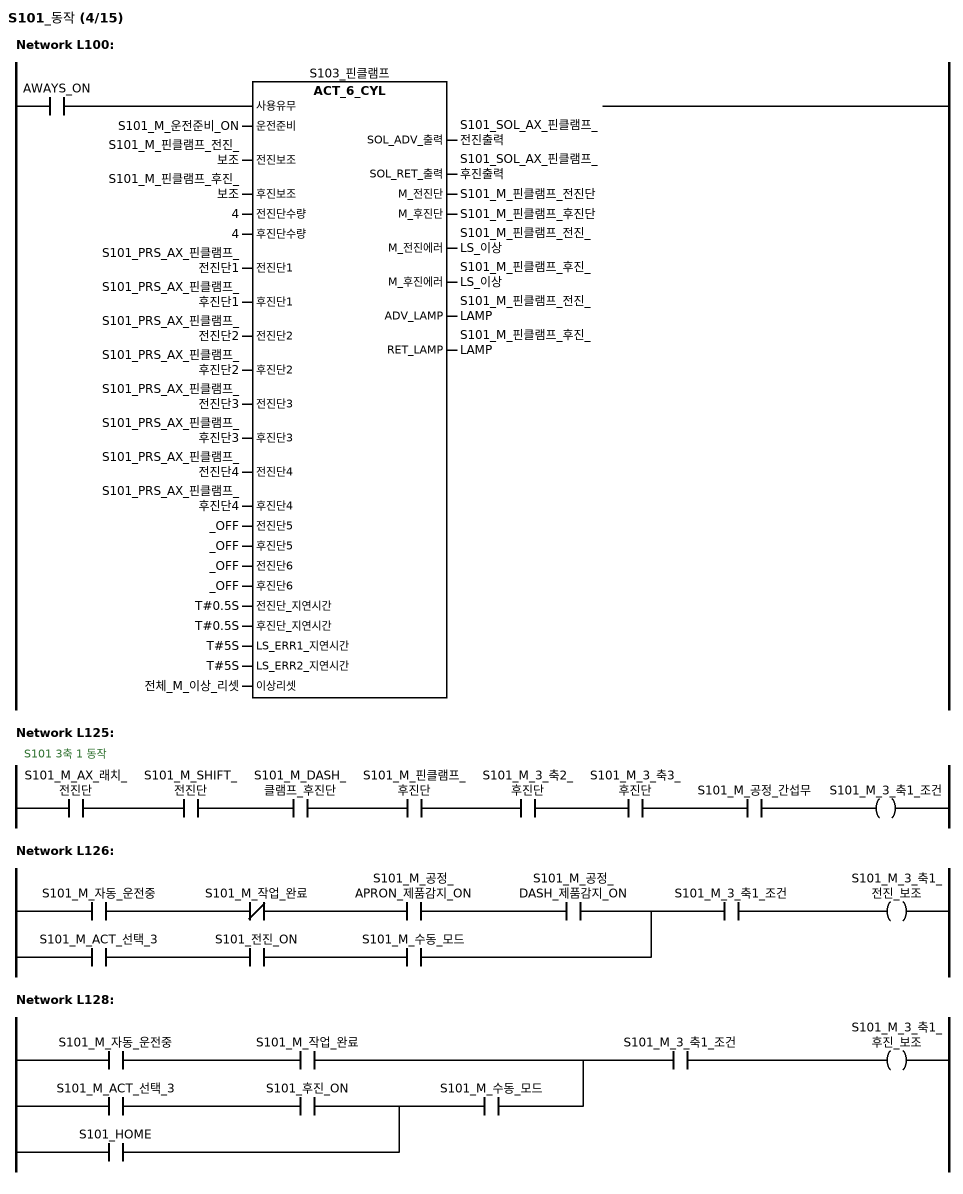
(* Rung L100 *)
S103_핀클램프(사용유무 := AWAYS_ON, 운전준비 := S101_M_운전준비_ON, 전진보조 := S101_M_핀클램프_전진_보조, 후진보조 := S101_M_핀클램프_후진_보조, 전진단수량 := 4, 후진단수량 := 4, 전진단1 := S101_PRS_AX_핀클램프_전진단1, 후진단1 := S101_PRS_AX_핀클램프_후진단1, 전진단2 := S101_PRS_AX_핀클램프_전진단2, 후진단2 := S101_PRS_AX_핀클램프_후진단2, 전진단3 := S101_PRS_AX_핀클램프_전진단3, 후진단3 := S101_PRS_AX_핀클램프_후진단3, 전진단4 := S101_PRS_AX_핀클램프_전진단4, 후진단4 := S101_PRS_AX_핀클램프_후진단4, 전진단5 := _OFF, 후진단5 := _OFF, 전진단6 := _OFF, 후진단6 := _OFF, 전진단_지연시간 := T#0.5S, 후진단_지연시간 := T#0.5S, LS_ERR1_지연시간 := T#5S, LS_ERR2_지연시간 := T#5S, 이상리셋 := 전체_M_이상_리셋, SOL_ADV_출력 => S101_SOL_AX_핀클램프_전진출력, SOL_RET_출력 => S101_SOL_AX_핀클램프_후진출력, M_전진단 => S101_M_핀클램프_전진단, M_후진단 => S101_M_핀클램프_후진단, M_전진에러 => S101_M_핀클램프_전진_LS_이상, M_후진에러 => S101_M_핀클램프_후진_LS_이상, ADV_LAMP => S101_M_핀클램프_전진_LAMP, RET_LAMP => S101_M_핀클램프_후진_LAMP);
(* S101 3축 1 동작 *)
(* Rung L125 *)
S101_M_3_축1_조건 := S101_M_AX_래치_전진단 AND S101_M_SHIFT_전진단 AND S101_M_DASH_클램프_후진단 AND S101_M_핀클램프_후진단 AND S101_M_3_축2_후진단 AND S101_M_3_축3_후진단 AND S101_M_공정_간섭무;
(* Rung L126 *)
S101_M_3_축1_전진_보조 := ((S101_M_자동_운전중 AND NOT S101_M_작업_완료 AND S101_M_공정_APRON_제품감지_ON AND S101_M_공정_DASH_제품감지_ON) OR (S101_M_ACT_선택_3 AND S101_전진_ON AND S101_M_수동_모드)) AND S101_M_3_축1_조건;
(* Rung L128 *)
S101_M_3_축1_후진_보조 := ((S101_M_자동_운전중 AND S101_M_작업_완료) OR (((S101_M_ACT_선택_3 AND S101_후진_ON) OR S101_HOME) AND S101_M_수동_모드)) AND S101_M_3_축1_조건;

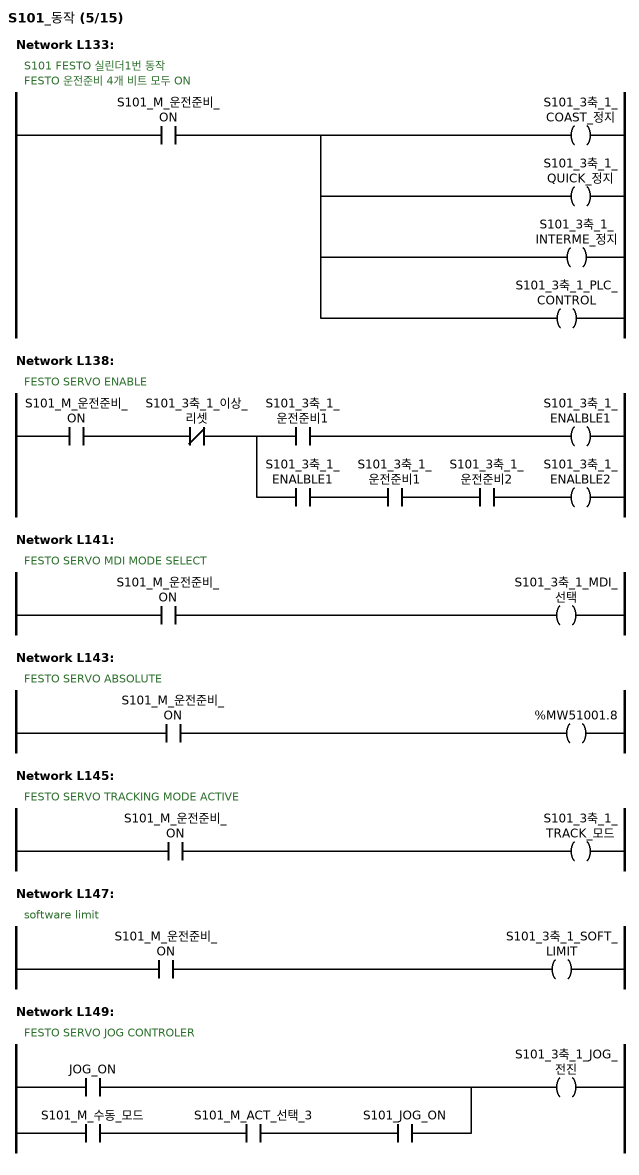
(* S101 FESTO 실린더1번 동작 *)
(* FESTO 운전준비 4개 비트 모두 ON *)
(* Rung L133 *)
S101_3축_1_COAST_정지 := S101_M_운전준비_ON;
S101_3축_1_QUICK_정지 := S101_M_운전준비_ON;
S101_3축_1_INTERME_정지 := S101_M_운전준비_ON;
S101_3축_1_PLC_CONTROL := S101_M_운전준비_ON;
(* FESTO SERVO ENABLE *)
(* Rung L138 *)
S101_3축_1_ENALBLE1 := S101_M_운전준비_ON AND NOT S101_3축_1_이상_리셋 AND S101_3축_1_운전준비1;
S101_3축_1_ENALBLE2 := S101_M_운전준비_ON AND NOT S101_3축_1_이상_리셋 AND S101_3축_1_ENALBLE1 AND S101_3축_1_운전준비1 AND S101_3축_1_운전준비2;
(* FESTO SERVO MDI MODE SELECT *)
(* Rung L141 *)
S101_3축_1_MDI_선택 := S101_M_운전준비_ON;
(* FESTO SERVO ABSOLUTE *)
(* Rung L143 *)
%MW51001.8 := S101_M_운전준비_ON;
(* FESTO SERVO TRACKING MODE ACTIVE *)
(* Rung L145 *)
S101_3축_1_TRACK_모드 := S101_M_운전준비_ON;
(* software limit *)
(* Rung L147 *)
S101_3축_1_SOFT_LIMIT := S101_M_운전준비_ON;
(* FESTO SERVO JOG CONTROLER *)
(* Rung L149 *)
S101_3축_1_JOG_전진 := JOG_ON OR (S101_M_수동_모드 AND S101_M_ACT_선택_3 AND S101_JOG_ON);

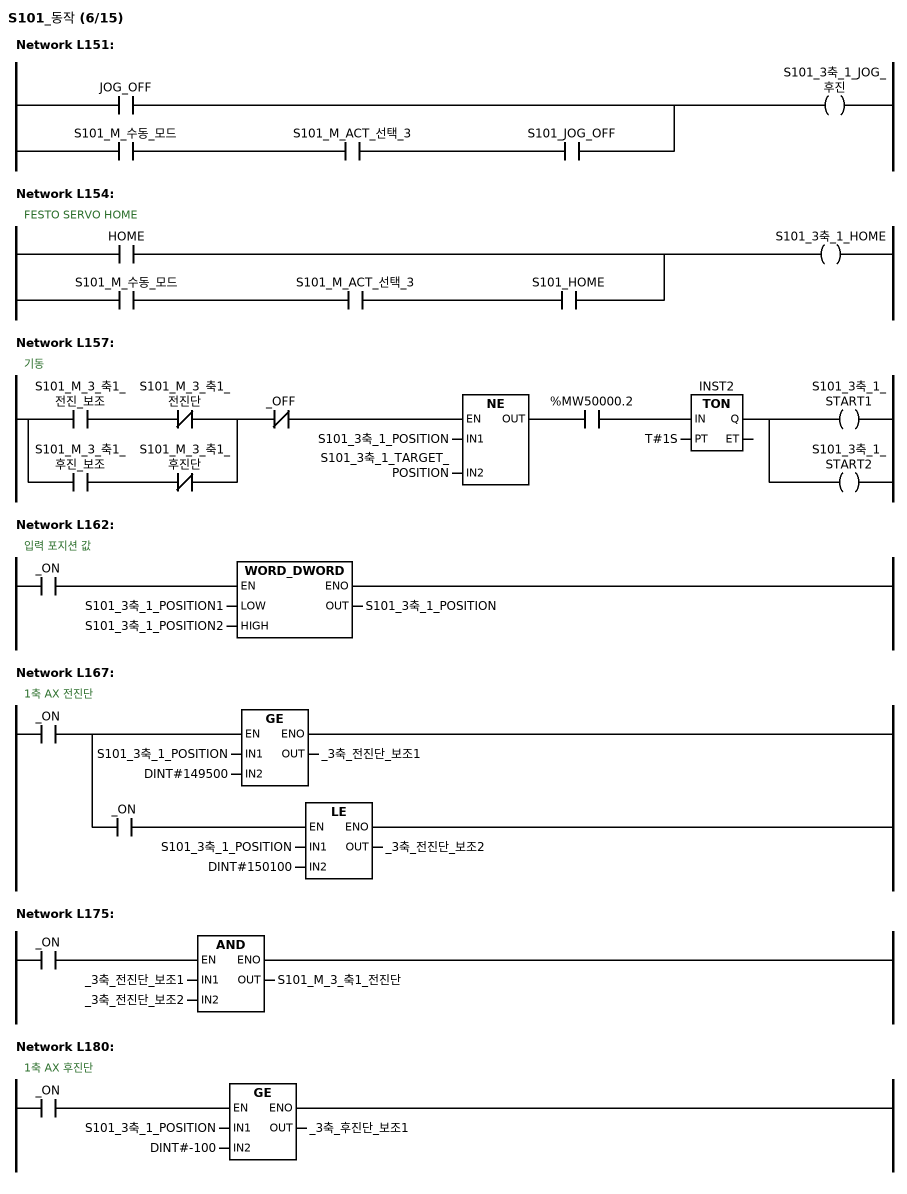
(* Rung L151 *)
S101_3축_1_JOG_후진 := JOG_OFF OR (S101_M_수동_모드 AND S101_M_ACT_선택_3 AND S101_JOG_OFF);
(* FESTO SERVO HOME *)
(* Rung L154 *)
S101_3축_1_HOME := HOME OR (S101_M_수동_모드 AND S101_M_ACT_선택_3 AND S101_HOME);
(* 기동 *)
(* Rung L157 *)
IF ((S101_M_3_축1_전진_보조 AND NOT S101_M_3_축1_전진단) OR (S101_M_3_축1_후진_보조 AND NOT S101_M_3_축1_후진단)) AND NOT _OFF THEN
    _t1 := S101_3축_1_POSITION <> S101_3축_1_TARGET_POSITION;
END_IF;
INST2(IN := _t1 AND %MW50000.2, PT := T#1S);
S101_3축_1_START1 := INST2.Q;
S101_3축_1_START2 := INST2.Q;
(* 입력 포지션 값 *)
(* Rung L162 *)
IF _ON THEN
    S101_3축_1_POSITION := WORD_DWORD(LOW := S101_3축_1_POSITION1, HIGH := S101_3축_1_POSITION2);
END_IF;
(* 1축 AX 전진단 *)
(* Rung L167 *)
IF _ON THEN _3축_전진단_보조1 := S101_3축_1_POSITION >= DINT#149500; END_IF;
IF _ON AND _ON THEN _3축_전진단_보조2 := S101_3축_1_POSITION <= DINT#150100; END_IF;
(* Rung L175 *)
IF _ON THEN S101_M_3_축1_전진단 := _3축_전진단_보조1 AND _3축_전진단_보조2; END_IF;
(* 1축 AX 후진단 *)
(* Rung L180 *)
IF _ON THEN _3축_후진단_보조1 := S101_3축_1_POSITION >= (DINT#-100); END_IF;

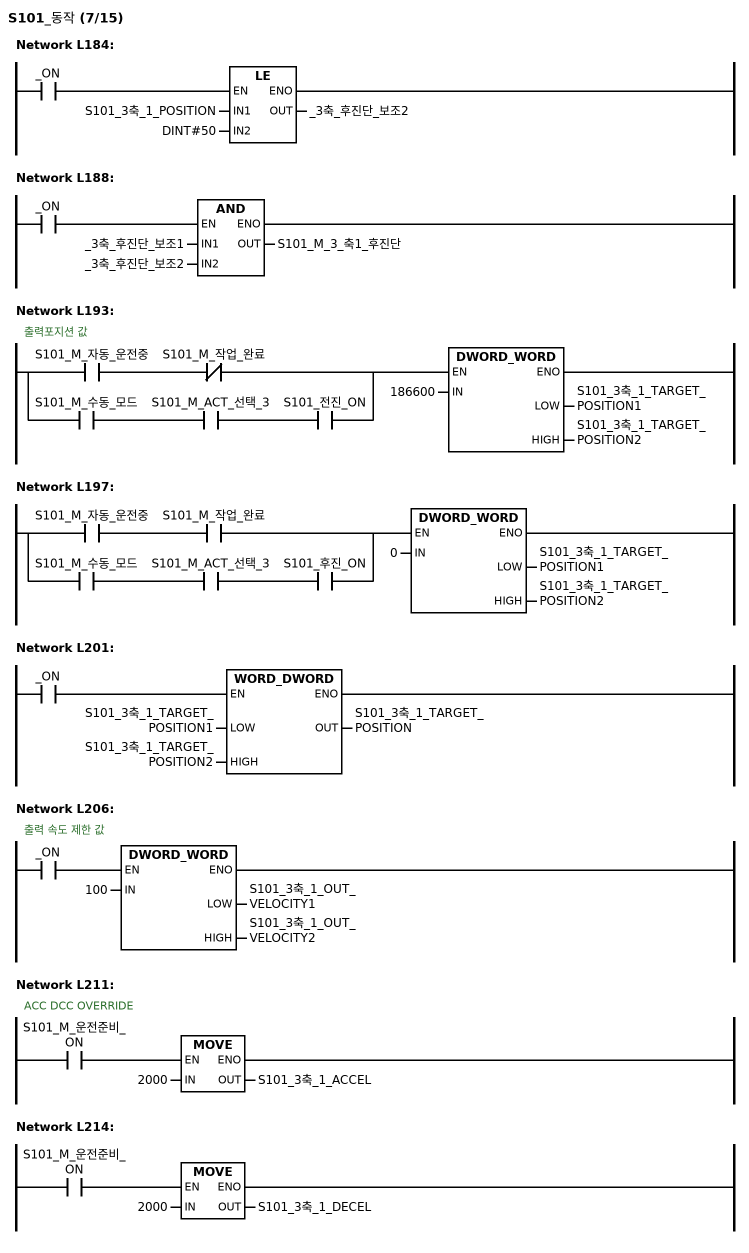
(* Rung L184 *)
IF _ON THEN _3축_후진단_보조2 := S101_3축_1_POSITION <= DINT#50; END_IF;
(* Rung L188 *)
IF _ON THEN S101_M_3_축1_후진단 := _3축_후진단_보조1 AND _3축_후진단_보조2; END_IF;
(* 출력포지션 값 *)
(* Rung L193 *)
IF (S101_M_자동_운전중 AND NOT S101_M_작업_완료) OR (S101_M_수동_모드 AND S101_M_ACT_선택_3 AND S101_전진_ON) THEN
    S101_3축_1_TARGET_POSITION1 := DWORD_WORD(IN := 186600, HIGH => S101_3축_1_TARGET_POSITION2);
END_IF;
(* Rung L197 *)
IF (S101_M_자동_운전중 AND S101_M_작업_완료) OR (S101_M_수동_모드 AND S101_M_ACT_선택_3 AND S101_후진_ON) THEN
    S101_3축_1_TARGET_POSITION1 := DWORD_WORD(IN := 0, HIGH => S101_3축_1_TARGET_POSITION2);
END_IF;
(* Rung L201 *)
IF _ON THEN
    S101_3축_1_TARGET_POSITION := WORD_DWORD(LOW := S101_3축_1_TARGET_POSITION1, HIGH := S101_3축_1_TARGET_POSITION2);
END_IF;
(* 출력 속도 제한 값 *)
(* Rung L206 *)
IF _ON THEN S101_3축_1_OUT_VELOCITY1 := DWORD_WORD(IN := 100, HIGH => S101_3축_1_OUT_VELOCITY2); END_IF;
(* ACC DCC OVERRIDE *)
(* Rung L211 *)
IF S101_M_운전준비_ON THEN S101_3축_1_ACCEL := 2000; END_IF;
(* Rung L214 *)
IF S101_M_운전준비_ON THEN S101_3축_1_DECEL := 2000; END_IF;

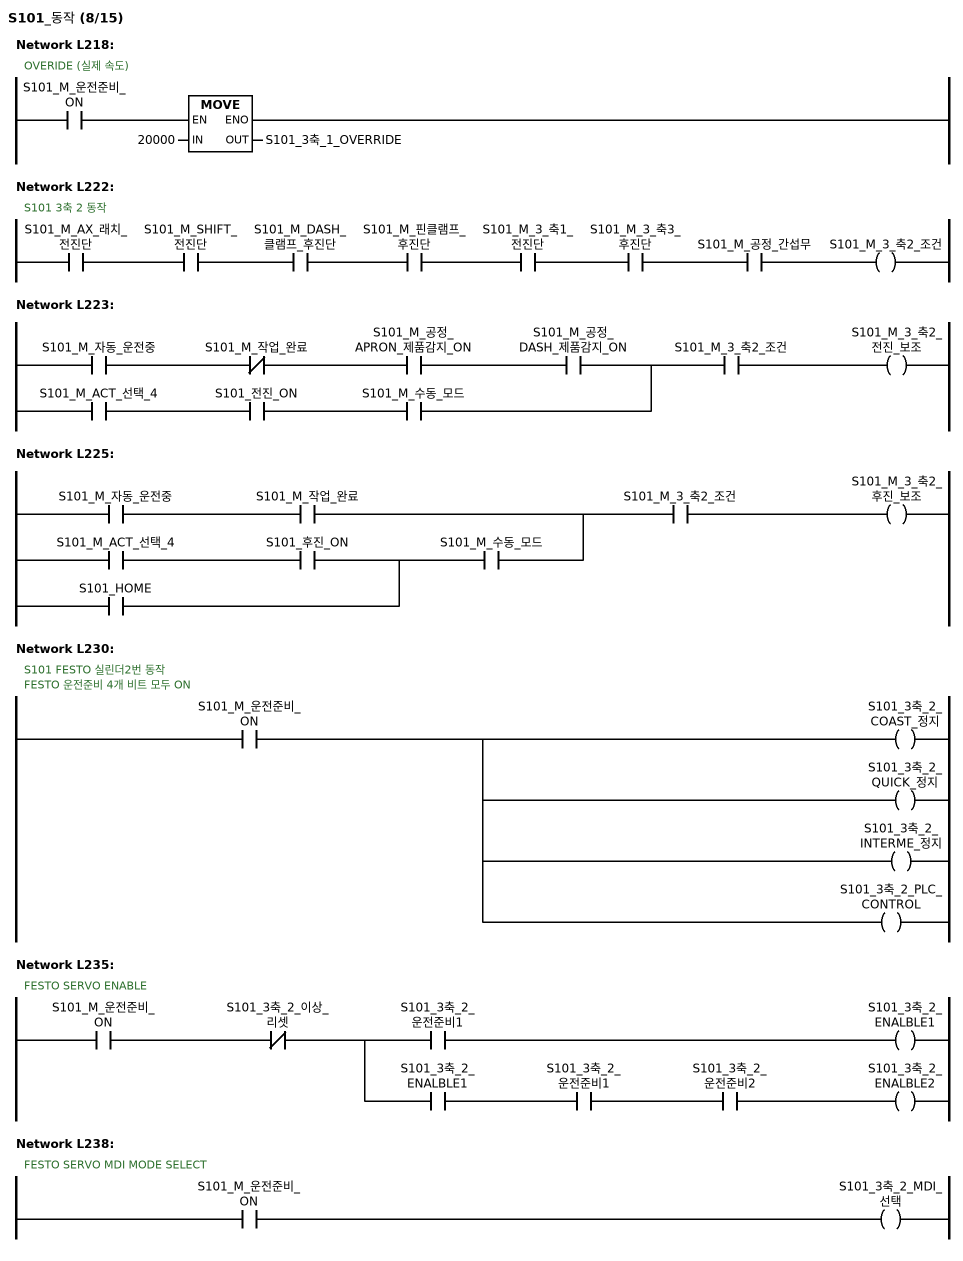
(* OVERIDE (실제 속도) *)
(* Rung L218 *)
IF S101_M_운전준비_ON THEN S101_3축_1_OVERRIDE := 20000; END_IF;
(* S101 3축 2 동작 *)
(* Rung L222 *)
S101_M_3_축2_조건 := S101_M_AX_래치_전진단 AND S101_M_SHIFT_전진단 AND S101_M_DASH_클램프_후진단 AND S101_M_핀클램프_후진단 AND S101_M_3_축1_전진단 AND S101_M_3_축3_후진단 AND S101_M_공정_간섭무;
(* Rung L223 *)
S101_M_3_축2_전진_보조 := ((S101_M_자동_운전중 AND NOT S101_M_작업_완료 AND S101_M_공정_APRON_제품감지_ON AND S101_M_공정_DASH_제품감지_ON) OR (S101_M_ACT_선택_4 AND S101_전진_ON AND S101_M_수동_모드)) AND S101_M_3_축2_조건;
(* Rung L225 *)
S101_M_3_축2_후진_보조 := ((S101_M_자동_운전중 AND S101_M_작업_완료) OR (((S101_M_ACT_선택_4 AND S101_후진_ON) OR S101_HOME) AND S101_M_수동_모드)) AND S101_M_3_축2_조건;
(* S101 FESTO 실린더2번 동작 *)
(* FESTO 운전준비 4개 비트 모두 ON *)
(* Rung L230 *)
S101_3축_2_COAST_정지 := S101_M_운전준비_ON;
S101_3축_2_QUICK_정지 := S101_M_운전준비_ON;
S101_3축_2_INTERME_정지 := S101_M_운전준비_ON;
S101_3축_2_PLC_CONTROL := S101_M_운전준비_ON;
(* FESTO SERVO ENABLE *)
(* Rung L235 *)
S101_3축_2_ENALBLE1 := S101_M_운전준비_ON AND NOT S101_3축_2_이상_리셋 AND S101_3축_2_운전준비1;
S101_3축_2_ENALBLE2 := S101_M_운전준비_ON AND NOT S101_3축_2_이상_리셋 AND S101_3축_2_ENALBLE1 AND S101_3축_2_운전준비1 AND S101_3축_2_운전준비2;
(* FESTO SERVO MDI MODE SELECT *)
(* Rung L238 *)
S101_3축_2_MDI_선택 := S101_M_운전준비_ON;

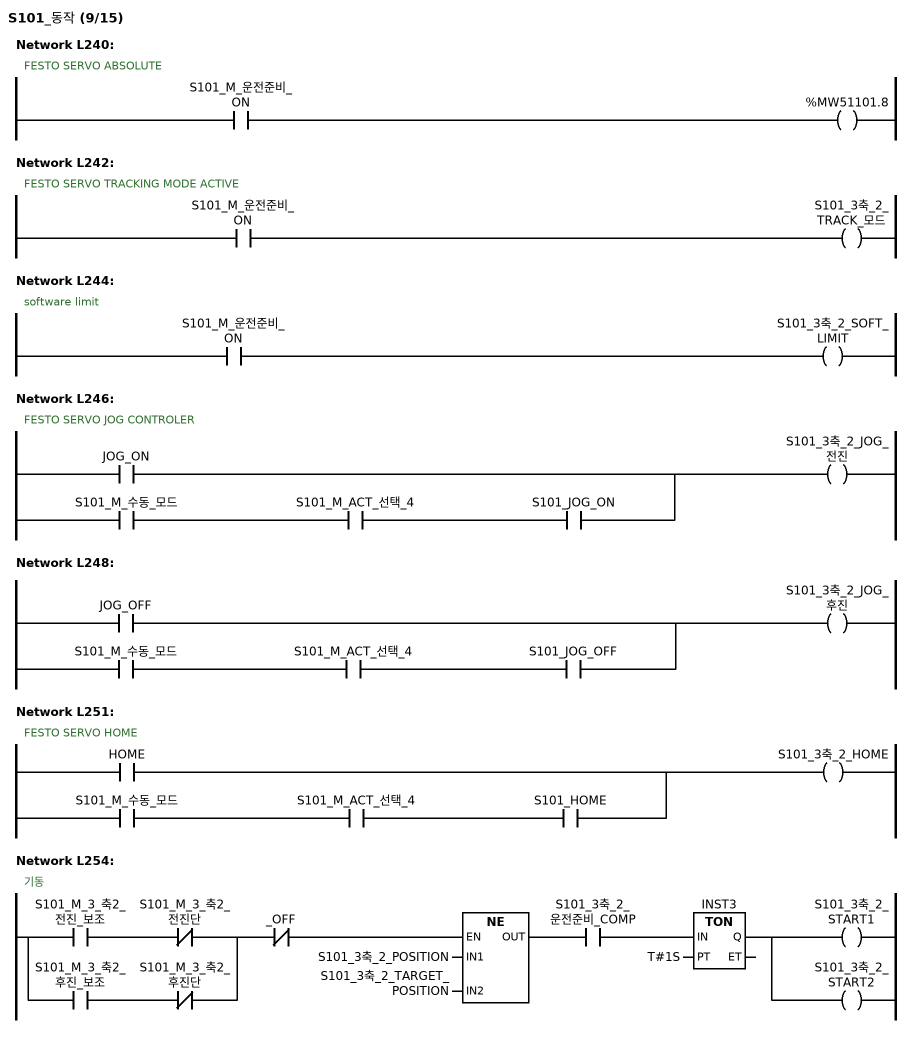
(* FESTO SERVO ABSOLUTE *)
(* Rung L240 *)
%MW51101.8 := S101_M_운전준비_ON;
(* FESTO SERVO TRACKING MODE ACTIVE *)
(* Rung L242 *)
S101_3축_2_TRACK_모드 := S101_M_운전준비_ON;
(* software limit *)
(* Rung L244 *)
S101_3축_2_SOFT_LIMIT := S101_M_운전준비_ON;
(* FESTO SERVO JOG CONTROLER *)
(* Rung L246 *)
S101_3축_2_JOG_전진 := JOG_ON OR (S101_M_수동_모드 AND S101_M_ACT_선택_4 AND S101_JOG_ON);
(* Rung L248 *)
S101_3축_2_JOG_후진 := JOG_OFF OR (S101_M_수동_모드 AND S101_M_ACT_선택_4 AND S101_JOG_OFF);
(* FESTO SERVO HOME *)
(* Rung L251 *)
S101_3축_2_HOME := HOME OR (S101_M_수동_모드 AND S101_M_ACT_선택_4 AND S101_HOME);
(* 기동 *)
(* Rung L254 *)
IF ((S101_M_3_축2_전진_보조 AND NOT S101_M_3_축2_전진단) OR (S101_M_3_축2_후진_보조 AND NOT S101_M_3_축2_후진단)) AND NOT _OFF THEN
    _t2 := S101_3축_2_POSITION <> S101_3축_2_TARGET_POSITION;
END_IF;
INST3(IN := _t2 AND S101_3축_2_운전준비_COMP, PT := T#1S);
S101_3축_2_START1 := INST3.Q;
S101_3축_2_START2 := INST3.Q;

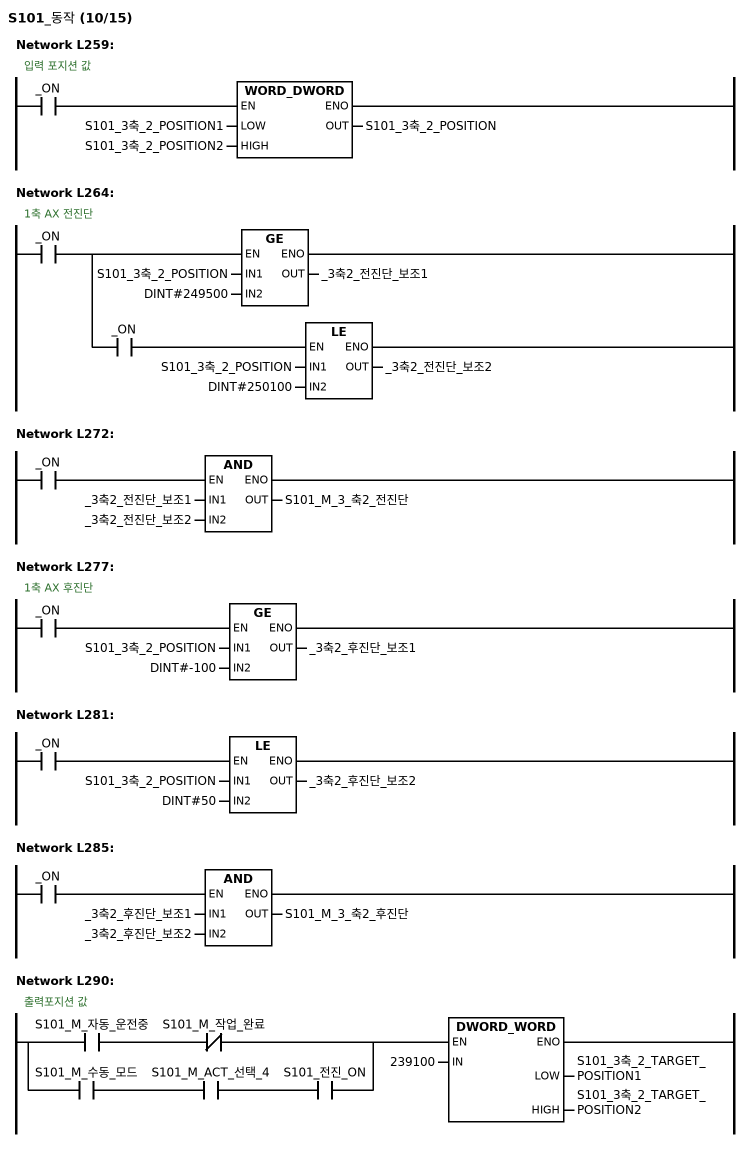
(* 입력 포지션 값 *)
(* Rung L259 *)
IF _ON THEN
    S101_3축_2_POSITION := WORD_DWORD(LOW := S101_3축_2_POSITION1, HIGH := S101_3축_2_POSITION2);
END_IF;
(* 1축 AX 전진단 *)
(* Rung L264 *)
IF _ON THEN _3축2_전진단_보조1 := S101_3축_2_POSITION >= DINT#249500; END_IF;
IF _ON AND _ON THEN _3축2_전진단_보조2 := S101_3축_2_POSITION <= DINT#250100; END_IF;
(* Rung L272 *)
IF _ON THEN S101_M_3_축2_전진단 := _3축2_전진단_보조1 AND _3축2_전진단_보조2; END_IF;
(* 1축 AX 후진단 *)
(* Rung L277 *)
IF _ON THEN _3축2_후진단_보조1 := S101_3축_2_POSITION >= (DINT#-100); END_IF;
(* Rung L281 *)
IF _ON THEN _3축2_후진단_보조2 := S101_3축_2_POSITION <= DINT#50; END_IF;
(* Rung L285 *)
IF _ON THEN S101_M_3_축2_후진단 := _3축2_후진단_보조1 AND _3축2_후진단_보조2; END_IF;
(* 출력포지션 값 *)
(* Rung L290 *)
IF (S101_M_자동_운전중 AND NOT S101_M_작업_완료) OR (S101_M_수동_모드 AND S101_M_ACT_선택_4 AND S101_전진_ON) THEN
    S101_3축_2_TARGET_POSITION1 := DWORD_WORD(IN := 239100, HIGH => S101_3축_2_TARGET_POSITION2);
END_IF;

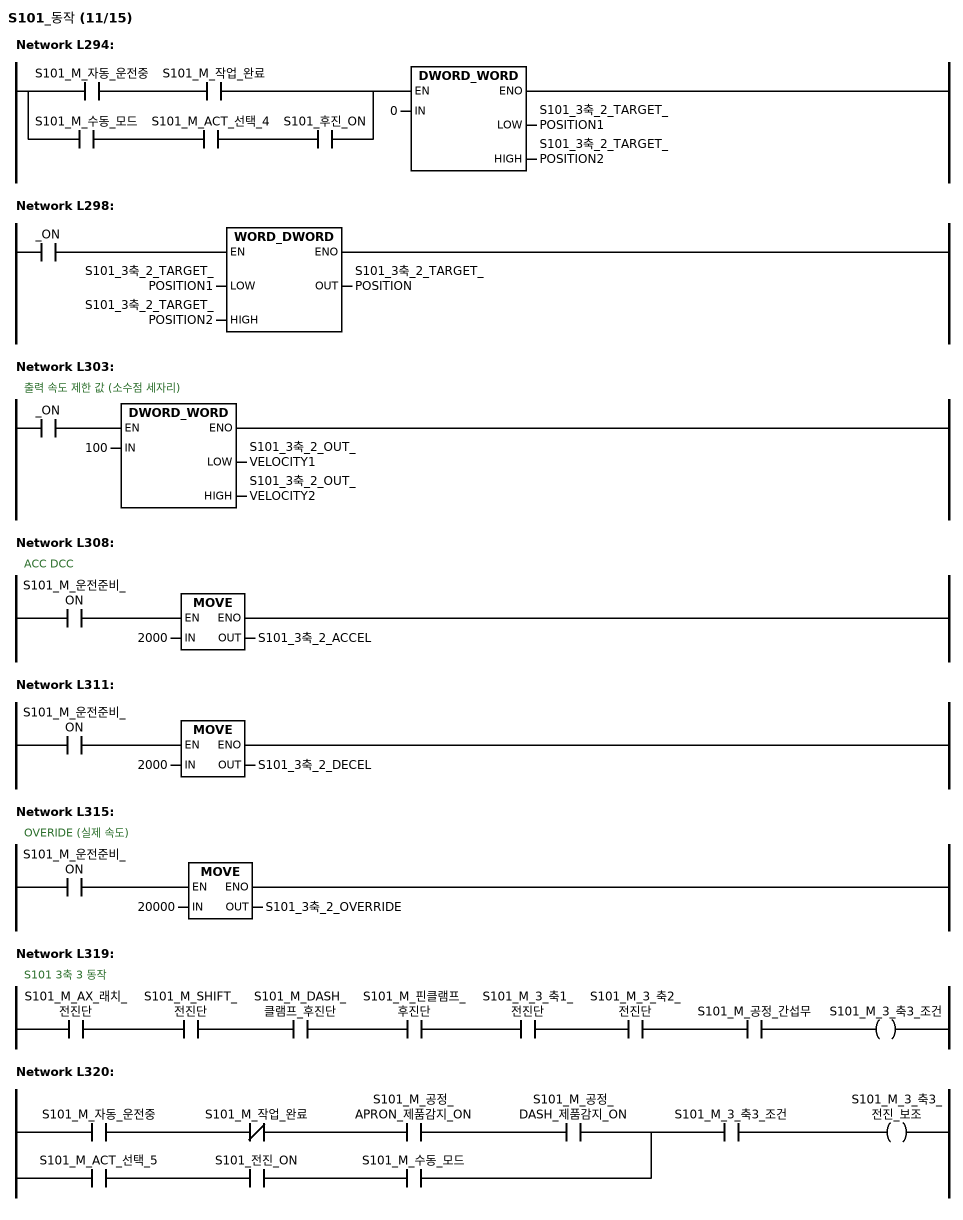
(* Rung L294 *)
IF (S101_M_자동_운전중 AND S101_M_작업_완료) OR (S101_M_수동_모드 AND S101_M_ACT_선택_4 AND S101_후진_ON) THEN
    S101_3축_2_TARGET_POSITION1 := DWORD_WORD(IN := 0, HIGH => S101_3축_2_TARGET_POSITION2);
END_IF;
(* Rung L298 *)
IF _ON THEN
    S101_3축_2_TARGET_POSITION := WORD_DWORD(LOW := S101_3축_2_TARGET_POSITION1, HIGH := S101_3축_2_TARGET_POSITION2);
END_IF;
(* 출력 속도 제한 값 (소수점 세자리) *)
(* Rung L303 *)
IF _ON THEN S101_3축_2_OUT_VELOCITY1 := DWORD_WORD(IN := 100, HIGH => S101_3축_2_OUT_VELOCITY2); END_IF;
(* ACC DCC *)
(* Rung L308 *)
IF S101_M_운전준비_ON THEN S101_3축_2_ACCEL := 2000; END_IF;
(* Rung L311 *)
IF S101_M_운전준비_ON THEN S101_3축_2_DECEL := 2000; END_IF;
(* OVERIDE (실제 속도) *)
(* Rung L315 *)
IF S101_M_운전준비_ON THEN S101_3축_2_OVERRIDE := 20000; END_IF;
(* S101 3축 3 동작 *)
(* Rung L319 *)
S101_M_3_축3_조건 := S101_M_AX_래치_전진단 AND S101_M_SHIFT_전진단 AND S101_M_DASH_클램프_후진단 AND S101_M_핀클램프_후진단 AND S101_M_3_축1_전진단 AND S101_M_3_축2_전진단 AND S101_M_공정_간섭무;
(* Rung L320 *)
S101_M_3_축3_전진_보조 := ((S101_M_자동_운전중 AND NOT S101_M_작업_완료 AND S101_M_공정_APRON_제품감지_ON AND S101_M_공정_DASH_제품감지_ON) OR (S101_M_ACT_선택_5 AND S101_전진_ON AND S101_M_수동_모드)) AND S101_M_3_축3_조건;

